LIN {X 0,Y 122.45,Z 109.011,A -85,B 0,C 180,E1 -25952.066,E2 -25952.066} C_VEL
LIN {X 0,Y 126.143,Z 114.519,A -85,B 0,C 180,E1 -25954.582,E2 -25954.582} C_VEL
LIN {X 0,Y 129.756,Z 120.065,A -85,B 0,C 180,E1 -25956.81,E2 -25956.81} C_VEL
LIN {X 0,Y 134.264,Z 129.772,A -85,B 0,C 180,E1 -25959.517,E2 -25959.517} C_VEL
LIN {X 0,Y 138.304,Z 140.286,A -85,B 0,C 180,E1 -25961.832,E2 -25961.832} C_VEL
LIN {X 0,Y 140.231,Z 146.487,A -85,B 0,C 180,E1 -25962.943,E2 -25962.943} C_VEL
LIN {X 0,Y 141.292,Z 167.319,A -85,B 0,C 180,E1 -25964.672,E2 -25964.672} C_VEL
LIN {X 0,Y 138.783,Z 203.821,A -85,B 0,C 180,E1 -25966.343,E2 -25966.343} C_VEL
LIN {X 0,Y 136.982,Z 217.471,A -85,B 0,C 180,E1 -25967.481,E2 -25967.481} C_VEL
LIN {X 0,Y 134.526,Z 229.675,A -85,B 0,C 180,E1 -25968.981,E2 -25968.981} C_VEL
LIN {X 0,Y 131.446,Z 241.678,A -85,B 0,C 180,E1 -25971.079,E2 -25971.079} C_VEL
LIN {X 0,Y 127.778,Z 253.16,A -85,B 0,C 180,E1 -25973.752,E2 -25973.752} C_VEL
LIN {X 0,Y 124.606,Z 262.476,A -85,B 0,C 180,E1 -25976.637,E2 -25976.637} C_VEL
LIN {X 0,Y 121.036,Z 272.287,A -85,B 0,C 180,E1 -25980.572,E2 -25980.572} C_VEL
LIN {X 0,Y 118.688,Z 278.374,A -85,B 0,C 180,E1 -25983.633,E2 -25983.633} C_VEL
LIN {X 0,Y 115.905,Z 286.343,A -85,B 0,C 180,E1 -25988.664,E2 -25988.664} C_VEL
LIN {X 0,Y 113.859,Z 292.673,A -85,B 0,C 180,E1 -25993.872,E2 -25993.872} C_VEL
LIN {X 0,Y 112.784,Z 297.7,A -85,B 0,C 180,E1 -25999.224,E2 -25999.224} C_VEL
LIN {X 0,Y 112.572,Z 301.563,A -85,B 0,C 180,E1 -26004.625,E2 -26004.625} C_VEL
LIN {X 0,Y 112.803,Z 304.341,A -85,B 0,C 180,E1 -26009.999,E2 -26009.999} C_VEL
LIN {X 0,Y 112.582,Z 305.583,A -85,B 0,C 180,E1 -26013.578,E2 -26013.578} C_VEL
LIN {X 0,Y 112.809,Z 306.873,A -85,B 0,C 180,E1 -26020.771,E2 -26020.771} C_VEL
LIN {X 0,Y 114.614,Z 306.557,A -85,B 0,C 180,E1 -26027.853,E2 -26027.853} C_VEL
LIN {X 0,Y 118.283,Z 304.747,A -85,B 0,C 180,E1 -26034.576,E2 -26034.576} C_VEL
LIN {X 0,Y 120.676,Z 303.239,A -85,B 0,C 180,E1 -26037.768,E2 -26037.768} C_VEL
LIN {X 0,Y 125.854,Z 299.488,A -85,B 0,C 180,E1 -26043.109,E2 -26043.109} C_VEL
LIN {X 0,Y 131.819,Z 294.518,A -85,B 0,C 180,E1 -26047.814,E2 -26047.814} C_VEL
LIN {X 0,Y 137.879,Z 288.943,A -85,B 0,C 180,E1 -26051.5,E2 -26051.5} C_VEL
LIN {X 0,Y 144.484,Z 282.029,A -85,B 0,C 180,E1 -26054.853,E2 -26054.853} C_VEL
LIN {X 0,Y 150.329,Z 275.005,A -85,B 0,C 180,E1 -26057.418,E2 -26057.418} C_VEL
LIN {X 0,Y 153.184,Z 271.302,A -85,B 0,C 180,E1 -26058.5,E2 -26058.5} C_VEL
LIN {X 0,Y 155.841,Z 267.217,A -85,B 0,C 180,E1 -26059.737,E2 -26059.737} C_VEL
LIN {X 0,Y 158.817,Z 260.366,A -85,B 0,C 180,E1 -26062.115,E2 -26062.115} C_VEL
LIN {X 0,Y 161.563,Z 253.029,A -85,B 0,C 180,E1 -26064.286,E2 -26064.286} C_VEL
LIN {X 0,Y 163.755,Z 248.186,A -85,B 0,C 180,E1 -26065.183,E2 -26065.183} C_VEL
LIN {X 0,Y 168.724,Z 237.706,A -85,B 0,C 180,E1 -26066.414,E2 -26066.414} C_VEL
LIN {X 0,Y 173.412,Z 225.079,A -85,B 0,C 180,E1 -26067.508,E2 -26067.508} C_VEL
LIN {X 0,Y 176.771,Z 212.767,A -85,B 0,C 180,E1 -26068.283,E2 -26068.283} C_VEL
LIN {X 0,Y 179.12,Z 199.548,A -85,B 0,C 180,E1 -26068.839,E2 -26068.839} C_VEL
LIN {X 0,Y 179.992,Z 191.121,A -85,B 0,C 180,E1 -26069.109,E2 -26069.109} C_VEL
LIN {X 0,Y 176.857,Z 181.807,A -85,B 0,C 180,E1 -26072.407,E2 -26072.407} C_VEL
LIN {X 0,Y 174.407,Z 175.318,A -85,B 0,C 180,E1 -26075.367,E2 -26075.367} C_VEL
LIN {X 0,Y 172.703,Z 171.191,A -85,B 0,C 180,E1 -26077.731,E2 -26077.731} C_VEL
LIN {X 0,Y 171.544,Z 168.304,A -85,B 0,C 180,E1 -26079.638,E2 -26079.638} C_VEL
LIN {X 0,Y 170.023,Z 164.562,A -85,B 0,C 180,E1 -26082.687,E2 -26082.687} C_VEL
LIN {X 0,Y 168.16,Z 160.166,A -85,B 0,C 180,E1 -26088.55,E2 -26088.55} C_VEL
LIN {X 0,Y 167.654,Z 159.81,A -85,B 0,C 180,E1 -26095.191,E2 -26095.191} C_VEL
LIN {X 0,Y 168.258,Z 159.961,A -85,B 0,C 180,E1 -26098.515,E2 -26098.515} C_VEL
LIN {X 0,Y 169.813,Z 163.596,A -85,B 0,C 180,E1 -26103.49,E2 -26103.49} C_VEL
LIN {X 0,Y 170.565,Z 164.869,A -85,B 0,C 180,E1 -26105.061,E2 -26105.061} C_VEL
LIN {X 0,Y 172.912,Z 169.191,A -85,B 0,C 180,E1 -26108.993,E2 -26108.993} C_VEL
LIN {X 0,Y 174.96,Z 172.997,A -85,B 0,C 180,E1 -26111.66,E2 -26111.66} C_VEL
LIN {X 0,Y 177.973,Z 178.76,A -85,B 0,C 180,E1 -26114.947,E2 -26114.947} C_VEL
LIN {X 0,Y 180.591,Z 184.208,A -85,B 0,C 180,E1 -26117.431,E2 -26117.431} C_VEL
LIN {X 0,Y 178.865,Z 198.313,A -85,B 0,C 180,E1 -26117.998,E2 -26117.998} C_VEL
LIN {X 0,Y 176.444,Z 209.589,A -85,B 0,C 180,E1 -26118.65,E2 -26118.65} C_VEL
LIN {X 0,Y 172.507,Z 222.682,A -85,B 0,C 180,E1 -26119.771,E2 -26119.771} C_VEL
LIN {X 0,Y 167.722,Z 234.725,A -85,B 0,C 180,E1 -26121.202,E2 -26121.202} C_VEL
LIN {X 0,Y 161.91,Z 246.089,A -85,B 0,C 180,E1 -26122.996,E2 -26122.996} C_VEL
LIN {X 0,Y 155.356,Z 256.599,A -85,B 0,C 180,E1 -26125.211,E2 -26125.211} C_VEL
LIN {X 0,Y 149.014,Z 265.155,A -85,B 0,C 180,E1 -26127.643,E2 -26127.643} C_VEL
LIN {X 0,Y 141.367,Z 273.791,A -85,B 0,C 180,E1 -26130.956,E2 -26130.956} C_VEL
LIN {X 0,Y 135.511,Z 279.488,A -85,B 0,C 180,E1 -26133.923,E2 -26133.923} C_VEL
LIN {X 0,Y 129.063,Z 284.989,A -85,B 0,C 180,E1 -26137.856,E2 -26137.856} C_VEL
LIN {X 0,Y 123.213,Z 289.225,A -85,B 0,C 180,E1 -26142.142,E2 -26142.142} C_VEL
LIN {X 0,Y 119.679,Z 291.431,A -85,B 0,C 180,E1 -26145.198,E2 -26145.198} C_VEL
LIN {X 0,Y 116.501,Z 293.121,A -85,B 0,C 180,E1 -26148.428,E2 -26148.428} C_VEL
LIN {X 0,Y 111.529,Z 295.153,A -85,B 0,C 180,E1 -26155.006,E2 -26155.006} C_VEL
LIN {X 0,Y 109.306,Z 295.609,A -85,B 0,C 180,E1 -26159.046,E2 -26159.046} C_VEL
LIN {X 0,Y 107.714,Z 295.578,A -85,B 0,C 180,E1 -26162.825,E2 -26162.825} C_VEL
LIN {X 0,Y 106.239,Z 294.936,A -85,B 0,C 180,E1 -26167.844,E2 -26167.844} C_VEL
LIN {X 0,Y 105.204,Z 293.009,A -85,B 0,C 180,E1 -26174.503,E2 -26174.503} C_VEL
LIN {X 0,Y 105.355,Z 290.275,A -85,B 0,C 180,E1 -26180.401,E2 -26180.401} C_VEL
LIN {X 0,Y 106.271,Z 286.516,A -85,B 0,C 180,E1 -26186.209,E2 -26186.209} C_VEL
LIN {X 0,Y 107.818,Z 281.647,A -85,B 0,C 180,E1 -26191.869,E2 -26191.869} C_VEL
LIN {X 0,Y 110.085,Z 275.523,A -85,B 0,C 180,E1 -26197.337,E2 -26197.337} C_VEL
LIN {X 0,Y 113.199,Z 267.91,A -85,B 0,C 180,E1 -26202.552,E2 -26202.552} C_VEL
LIN {X 0,Y 116.412,Z 260.121,A -85,B 0,C 180,E1 -26206.666,E2 -26206.666} C_VEL
LIN {X 0,Y 120.098,Z 250.61,A -85,B 0,C 180,E1 -26210.557,E2 -26210.557} C_VEL
LIN {X 0,Y 123.738,Z 240.071,A -85,B 0,C 180,E1 -26213.872,E2 -26213.872} C_VEL
LIN {X 0,Y 127.123,Z 228.378,A -85,B 0,C 180,E1 -26216.693,E2 -26216.693} C_VEL
LIN {X 0,Y 130.218,Z 215.809,A -85,B 0,C 180,E1 -26218.841,E2 -26218.841} C_VEL
LIN {X 0,Y 132.564,Z 202.695,A -85,B 0,C 180,E1 -26220.45,E2 -26220.45} C_VEL
LIN {X 0,Y 134.047,Z 189.846,A -85,B 0,C 180,E1 -26221.461,E2 -26221.461} C_VEL
LIN {X 0,Y 137.031,Z 146.864,A -85,B 0,C 180,E1 -26223.415,E2 -26223.415} C_VEL
LIN {X 0,Y 131.983,Z 135.808,A -85,B 0,C 180,E1 -26226.218,E2 -26226.218} C_VEL
LIN {X 0,Y 126.284,Z 125.434,A -85,B 0,C 180,E1 -26229.657,E2 -26229.657} C_VEL
LIN {X 0,Y 120.985,Z 117.374,A -85,B 0,C 180,E1 -26233.233,E2 -26233.233} C_VEL
LIN {X 0,Y 118.365,Z 113.693,A -85,B 0,C 180,E1 -26235.205,E2 -26235.205} C_VEL
LIN {X 0,Y 115.945,Z 110.284,A -85,B 0,C 180,E1 -26237.198,E2 -26237.198} C_VEL
LIN {X 0,Y 114.847,Z 109.03,A -85,B 0,C 180,E1 -26238.132,E2 -26238.132} C_VEL
LIN {X 0,Y 112.7,Z 106.255,A -85,B 0,C 180,E1 -26240.122,E2 -26240.122} C_VEL
LIN {X 0,Y 111.818,Z 104.593,A -85,B 0,C 180,E1 -26241.058,E2 -26241.058} C_VEL
LIN {X 0,Y 109.131,Z 102.466,A -85,B 0,C 180,E1 -26243.769,E2 -26243.769} C_VEL
LIN {X 0,Y 107.991,Z 100.283,A -85,B 0,C 180,E1 -26245.22,E2 -26245.22} C_VEL
LIN {X 0,Y 107.742,Z 98.998,A -85,B 0,C 180,E1 -26245.795,E2 -26245.795} C_VEL
LIN {X 0,Y 107.8,Z 99.021,A -85,B 0,C 180,E1 -26248.562,E2 -26248.562} C_VEL
LIN {X 0,Y 107.862,Z 99.029,A -85,B 0,C 180,E1 -26255.814,E2 -26255.814} C_VEL
LIN {X 0,Y 107.907,Z 99.037,A -85,B 0,C 180,E1 -26260.994,E2 -26260.994} C_VEL
LIN {X 0,Y 108.257,Z 98.997,A -85,B 0,C 180,E1 -26268.768,E2 -26268.768} C_VEL
LIN {X 0,Y 108.45,Z 98.975,A -85,B 0,C 180,E1 -26276.284,E2 -26276.284} C_VEL
LIN {X 0,Y 108.922,Z 98.897,A -85,B 0,C 180,E1 -26279.999,E2 -26279.999} C_VEL
LIN {X 0,Y 108.306,Z 98.976,A -85,B 0,C 180,E1 -26287.456,E2 -26287.456} C_VEL
LIN {X 0,Y 108.178,Z 99.006,A -85,B 0,C 180,E1 -26292.959,E2 -26292.959} C_VEL
LIN {X 0,Y 107.895,Z 99.064,A -85,B 0,C 180,E1 -26299.748,E2 -26299.748} C_VEL
LIN {X 0,Y 108.638,Z 101.364,A -85,B 0,C 180,E1 -26300.842,E2 -26300.842} C_VEL
LIN {X 0,Y 110.574,Z 103.726,A -85,B 0,C 180,E1 -26302.993,E2 -26302.993} C_VEL
LIN {X 0,Y 112.138,Z 104.975,A -85,B 0,C 180,E1 -26304.502,E2 -26304.502} C_VEL
LIN {X 0,Y 114.06,Z 108.164,A -85,B 0,C 180,E1 -26306.409,E2 -26306.409} C_VEL
LIN {X 0,Y 115.947,Z 110.168,A -85,B 0,C 180,E1 -26308.018,E2 -26308.018} C_VEL
LIN {X 0,Y 118.401,Z 113.66,A -85,B 0,C 180,E1 -26310.04,E2 -26310.04} C_VEL
LIN {X 0,Y 122.41,Z 119.495,A -85,B 0,C 180,E1 -26313.007,E2 -26313.007} C_VEL
LIN {X 0,Y 126.307,Z 125.87,A -85,B 0,C 180,E1 -26315.626,E2 -26315.626} C_VEL
LIN {X 0,Y 131.184,Z 137.371,A -85,B 0,C 180,E1 -26318.796,E2 -26318.796} C_VEL
LIN {X 0,Y 134.821,Z 148.268,A -85,B 0,C 180,E1 -26321.079,E2 -26321.079} C_VEL
LIN {X 0,Y 135.709,Z 164.102,A -85,B 0,C 180,E1 -26322.531,E2 -26322.531} C_VEL
LIN {X 0,Y 135.65,Z 169.911,A -85,B 0,C 180,E1 -26322.912,E2 -26322.912} C_VEL
LIN {X 0,Y 133.158,Z 204.005,A -85,B 0,C 180,E1 -26324.525,E2 -26324.525} C_VEL
LIN {X 0,Y 131.269,Z 217.462,A -85,B 0,C 180,E1 -26325.684,E2 -26325.684} C_VEL
LIN {X 0,Y 128.699,Z 229.567,A -85,B 0,C 180,E1 -26327.219,E2 -26327.219} C_VEL
LIN {X 0,Y 125.48,Z 241.506,A -85,B 0,C 180,E1 -26329.374,E2 -26329.374} C_VEL
LIN {X 0,Y 121.634,Z 252.948,A -85,B 0,C 180,E1 -26332.126,E2 -26332.126} C_VEL
LIN {X 0,Y 118.293,Z 262.236,A -85,B 0,C 180,E1 -26335.12,E2 -26335.12} C_VEL
LIN {X 0,Y 114.982,Z 270.896,A -85,B 0,C 180,E1 -26338.699,E2 -26338.699} C_VEL
LIN {X 0,Y 112.256,Z 277.325,A -85,B 0,C 180,E1 -26341.993,E2 -26341.993} C_VEL
LIN {X 0,Y 109.258,Z 285.443,A -85,B 0,C 180,E1 -26347.296,E2 -26347.296} C_VEL
LIN {X 0,Y 106.998,Z 291.889,A -85,B 0,C 180,E1 -26352.807,E2 -26352.807} C_VEL
LIN {X 0,Y 105.786,Z 297.003,A -85,B 0,C 180,E1 -26358.502,E2 -26358.502} C_VEL
LIN {X 0,Y 105.479,Z 300.944,A -85,B 0,C 180,E1 -26364.263,E2 -26364.263} C_VEL
LIN {X 0,Y 105.727,Z 303.8,A -85,B 0,C 180,E1 -26369.999,E2 -26369.999} C_VEL
LIN {X 0,Y 105.495,Z 305.076,A -85,B 0,C 180,E1 -26373.818,E2 -26373.818} C_VEL
LIN {X 0,Y 105.814,Z 306.437,A -85,B 0,C 180,E1 -26381.492,E2 -26381.492} C_VEL
LIN {X 0,Y 106.625,Z 306.536,A -85,B 0,C 180,E1 -26385.286,E2 -26385.286} C_VEL
LIN {X 0,Y 109.606,Z 305.539,A -85,B 0,C 180,E1 -26392.625,E2 -26392.625} C_VEL
LIN {X 0,Y 114.425,Z 303.036,A -85,B 0,C 180,E1 -26399.429,E2 -26399.429} C_VEL
LIN {X 0,Y 119.496,Z 299.708,A -85,B 0,C 180,E1 -26404.575,E2 -26404.575} C_VEL
LIN {X 0,Y 126.28,Z 294.491,A -85,B 0,C 180,E1 -26409.792,E2 -26409.792} C_VEL
LIN {X 0,Y 133.728,Z 287.998,A -85,B 0,C 180,E1 -26414.133,E2 -26414.133} C_VEL
LIN {X 0,Y 140.758,Z 280.932,A -85,B 0,C 180,E1 -26417.429,E2 -26417.429} C_VEL
LIN {X 0,Y 146.812,Z 273.785,A -85,B 0,C 180,E1 -26419.988,E2 -26419.988} C_VEL
LIN {X 0,Y 150.768,Z 268.778,A -85,B 0,C 180,E1 -26421.332,E2 -26421.332} C_VEL
LIN {X 0,Y 157.429,Z 259.05,A -85,B 0,C 180,E1 -26423.47,E2 -26423.47} C_VEL
LIN {X 0,Y 163.755,Z 248.186,A -85,B 0,C 180,E1 -26425.183,E2 -26425.183} C_VEL
LIN {X 0,Y 165.904,Z 243.232,A -85,B 0,C 180,E1 -26426.011,E2 -26426.011} C_VEL
LIN {X 0,Y 168.222,Z 234.981,A -85,B 0,C 180,E1 -26427.743,E2 -26427.743} C_VEL
LIN {X 0,Y 170.157,Z 226.466,A -85,B 0,C 180,E1 -26429.33,E2 -26429.33} C_VEL
LIN {X 0,Y 171.563,Z 221.002,A -85,B 0,C 180,E1 -26429.914,E2 -26429.914} C_VEL
LIN {X 0,Y 174.755,Z 208.28,A -85,B 0,C 180,E1 -26430.575,E2 -26430.575} C_VEL
LIN {X 0,Y 176.771,Z 195.011,A -85,B 0,C 180,E1 -26431.061,E2 -26431.061} C_VEL
LIN {X 0,Y 176.717,Z 193.931,A -85,B 0,C 180,E1 -26431.218,E2 -26431.218} C_VEL
LIN {X 0,Y 174.265,Z 186.165,A -85,B 0,C 180,E1 -26434.148,E2 -26434.148} C_VEL
LIN {X 0,Y 171.921,Z 179.559,A -85,B 0,C 180,E1 -26437.386,E2 -26437.386} C_VEL
LIN {X 0,Y 170.006,Z 174.486,A -85,B 0,C 180,E1 -26440.688,E2 -26440.688} C_VEL
LIN {X 0,Y 168.773,Z 171.173,A -85,B 0,C 180,E1 -26443.438,E2 -26443.438} C_VEL
LIN {X 0,Y 167.156,Z 167.137,A -85,B 0,C 180,E1 -26449.094,E2 -26449.094} C_VEL
LIN {X 0,Y 166.773,Z 166.854,A -85,B 0,C 180,E1 -26455.166,E2 -26455.166} C_VEL
LIN {X 0,Y 167.29,Z 167.015,A -85,B 0,C 180,E1 -26458.195,E2 -26458.195} C_VEL
LIN {X 0,Y 168.981,Z 170.859,A -85,B 0,C 180,E1 -26463.652,E2 -26463.652} C_VEL
LIN {X 0,Y 171.441,Z 175.774,A -85,B 0,C 180,E1 -26468.246,E2 -26468.246} C_VEL
LIN {X 0,Y 173.46,Z 179.789,A -85,B 0,C 180,E1 -26471.065,E2 -26471.065} C_VEL
LIN {X 0,Y 176.181,Z 185.405,A -85,B 0,C 180,E1 -26474.217,E2 -26474.217} C_VEL
LIN {X 0,Y 177.361,Z 187.99,A -85,B 0,C 180,E1 -26475.453,E2 -26475.453} C_VEL
LIN {X 0,Y 175.483,Z 200.905,A -85,B 0,C 180,E1 -26476.019,E2 -26476.019} C_VEL
LIN {X 0,Y 172.389,Z 213.819,A -85,B 0,C 180,E1 -26476.836,E2 -26476.836} C_VEL
LIN {X 0,Y 168.838,Z 224.584,A -85,B 0,C 180,E1 -26477.793,E2 -26477.793} C_VEL
LIN {X 0,Y 164.475,Z 235.023,A -85,B 0,C 180,E1 -26479.024,E2 -26479.024} C_VEL
LIN {X 0,Y 158.413,Z 246.497,A -85,B 0,C 180,E1 -26480.789,E2 -26480.789} C_VEL
LIN {X 0,Y 152.365,Z 255.923,A -85,B 0,C 180,E1 -26482.705,E2 -26482.705} C_VEL
LIN {X 0,Y 145.42,Z 265.067,A -85,B 0,C 180,E1 -26485.185,E2 -26485.185} C_VEL
LIN {X 0,Y 137.722,Z 273.511,A -85,B 0,C 180,E1 -26488.327,E2 -26488.327} C_VEL
LIN {X 0,Y 130.352,Z 280.348,A -85,B 0,C 180,E1 -26491.864,E2 -26491.864} C_VEL
LIN {X 0,Y 122.493,Z 286.54,A -85,B 0,C 180,E1 -26496.561,E2 -26496.561} C_VEL
LIN {X 0,Y 116.238,Z 290.588,A -85,B 0,C 180,E1 -26501.173,E2 -26501.173} C_VEL
LIN {X 0,Y 111.063,Z 293.32,A -85,B 0,C 180,E1 -26505.889,E2 -26505.889} C_VEL
LIN {X 0,Y 107.996,Z 294.627,A -85,B 0,C 180,E1 -26509.403,E2 -26509.403} C_VEL
LIN {X 0,Y 105.137,Z 295.571,A -85,B 0,C 180,E1 -26513.338,E2 -26513.338} C_VEL
LIN {X 0,Y 103.036,Z 295.986,A -85,B 0,C 180,E1 -26516.931,E2 -26516.931} C_VEL
LIN {X 0,Y 101.203,Z 295.999,A -85,B 0,C 180,E1 -26520.916,E2 -26520.916} C_VEL
LIN {X 0,Y 99.311,Z 295.302,A -85,B 0,C 180,E1 -26526.926,E2 -26526.926} C_VEL
LIN {X 0,Y 98.2,Z 293.605,A -85,B 0,C 180,E1 -26533.367,E2 -26533.367} C_VEL
LIN {X 0,Y 98.203,Z 290.964,A -85,B 0,C 180,E1 -26539.695,E2 -26539.695} C_VEL
LIN {X 0,Y 99.067,Z 287.302,A -85,B 0,C 180,E1 -26545.933,E2 -26545.933} C_VEL
LIN {X 0,Y 100.652,Z 282.536,A -85,B 0,C 180,E1 -26552.002,E2 -26552.002} C_VEL
LIN {X 0,Y 103.508,Z 275.394,A -85,B 0,C 180,E1 -26558.789,E2 -26558.789} C_VEL
LIN {X 0,Y 106.897,Z 267.646,A -85,B 0,C 180,E1 -26564.275,E2 -26564.275} C_VEL
LIN {X 0,Y 111.091,Z 257.912,A -85,B 0,C 180,E1 -26569.4,E2 -26569.4} C_VEL
LIN {X 0,Y 114.979,Z 248.275,A -85,B 0,C 180,E1 -26573.231,E2 -26573.231} C_VEL
LIN {X 0,Y 118.574,Z 237.94,A -85,B 0,C 180,E1 -26576.395,E2 -26576.395} C_VEL
LIN {X 0,Y 121.788,Z 227.166,A -85,B 0,C 180,E1 -26578.902,E2 -26578.902} C_VEL
LIN {X 0,Y 125.023,Z 214.295,A -85,B 0,C 180,E1 -26581.064,E2 -26581.064} C_VEL
LIN {X 0,Y 127.273,Z 201.737,A -85,B 0,C 180,E1 -26582.559,E2 -26582.559} C_VEL
LIN {X 0,Y 128.774,Z 188.552,A -85,B 0,C 180,E1 -26583.549,E2 -26583.549} C_VEL
LIN {X 0,Y 131.641,Z 149.15,A -85,B 0,C 180,E1 -26585.36,E2 -26585.36} C_VEL
LIN {X 0,Y 127.505,Z 139.82,A -85,B 0,C 180,E1 -26587.888,E2 -26587.888} C_VEL
LIN {X 0,Y 122.374,Z 130.243,A -85,B 0,C 180,E1 -26591.267,E2 -26591.267} C_VEL
LIN {X 0,Y 117.394,Z 122.443,A -85,B 0,C 180,E1 -26594.95,E2 -26594.95} C_VEL
LIN {X 0,Y 115.094,Z 119.173,A -85,B 0,C 180,E1 -26596.842,E2 -26596.842} C_VEL
LIN {X 0,Y 112.326,Z 115.229,A -85,B 0,C 180,E1 -26599.356,E2 -26599.356} C_VEL
LIN {X 0,Y 109.902,Z 111.933,A -85,B 0,C 180,E1 -26601.797,E2 -26601.797} C_VEL
LIN {X 0,Y 109.106,Z 110.795,A -85,B 0,C 180,E1 -26602.668,E2 -26602.668} C_VEL
LIN {X 0,Y 106.527,Z 108.161,A -85,B 0,C 180,E1 -26605.603,E2 -26605.603} C_VEL
LIN {X 0,Y 105.263,Z 105.654,A -85,B 0,C 180,E1 -26607.405,E2 -26607.405} C_VEL
LIN {X 0,Y 102.502,Z 103.847,A -85,B 0,C 180,E1 -26611.316,E2 -26611.316} C_VEL
LIN {X 0,Y 101.086,Z 101.44,A -85,B 0,C 180,E1 -26614.051,E2 -26614.051} C_VEL
LIN {X 0,Y 100.778,Z 99.911,A -85,B 0,C 180,E1 -26615.041,E2 -26615.041} C_VEL
LIN {X 0,Y 100.819,Z 99.927,A -85,B 0,C 180,E1 -26619.601,E2 -26619.601} C_VEL
LIN {X 0,Y 101.105,Z 99.885,A -85,B 0,C 180,E1 -26626.702,E2 -26626.702} C_VEL
LIN {X 0,Y 101.246,Z 99.851,A -85,B 0,C 180,E1 -26632.019,E2 -26632.019} C_VEL
LIN {X 0,Y 101.849,Z 99.777,A -85,B 0,C 180,E1 -26639.999,E2 -26639.999} C_VEL
LIN {X 0,Y 101.185,Z 99.869,A -85,B 0,C 180,E1 -26649.999,E2 -26649.999} C_VEL
LIN {X 0,Y 101.236,Z 100.081,A -85,B 0,C 180,E1 -26651.132,E2 -26651.132} C_VEL
LIN {X 0,Y 102.055,Z 102.596,A -85,B 0,C 180,E1 -26652.993,E2 -26652.993} C_VEL
LIN {X 0,Y 103.861,Z 104.818,A -85,B 0,C 180,E1 -26655.955,E2 -26655.955} C_VEL
LIN {X 0,Y 105.624,Z 105.943,A -85,B 0,C 180,E1 -26658.298,E2 -26658.298} C_VEL
LIN {X 0,Y 107.419,Z 109.132,A -85,B 0,C 180,E1 -26660.714,E2 -26660.714} C_VEL
LIN {X 0,Y 109.644,Z 111.32,A -85,B 0,C 180,E1 -26663.138,E2 -26663.138} C_VEL
LIN {X 0,Y 112.069,Z 114.908,A -85,B 0,C 180,E1 -26665.636,E2 -26665.636} C_VEL
LIN {X 0,Y 113.338,Z 116.523,A -85,B 0,C 180,E1 -26666.808,E2 -26666.808} C_VEL
LIN {X 0,Y 116.649,Z 121.303,A -85,B 0,C 180,E1 -26669.673,E2 -26669.673} C_VEL
LIN {X 0,Y 120.826,Z 127.796,A -85,B 0,C 180,E1 -26672.874,E2 -26672.874} C_VEL
LIN {X 0,Y 123.279,Z 132.744,A -85,B 0,C 180,E1 -26674.663,E2 -26674.663} C_VEL
LIN {X 0,Y 127.416,Z 143.33,A -85,B 0,C 180,E1 -26677.587,E2 -26677.587} C_VEL
LIN {X 0,Y 129.836,Z 151.229,A -85,B 0,C 180,E1 -26679.276,E2 -26679.276} C_VEL
LIN {X 0,Y 130.459,Z 168.381,A -85,B 0,C 180,E1 -26680.823,E2 -26680.823} C_VEL
LIN {X 0,Y 127.814,Z 203.093,A -85,B 0,C 180,E1 -26682.475,E2 -26682.475} C_VEL
LIN {X 0,Y 125.751,Z 217.127,A -85,B 0,C 180,E1 -26683.691,E2 -26683.691} C_VEL
LIN {X 0,Y 123.006,Z 229.451,A -85,B 0,C 180,E1 -26685.292,E2 -26685.292} C_VEL
LIN {X 0,Y 119.638,Z 241.334,A -85,B 0,C 180,E1 -26687.501,E2 -26687.501} C_VEL
LIN {X 0,Y 115.598,Z 252.736,A -85,B 0,C 180,E1 -26690.328,E2 -26690.328} C_VEL
LIN {X 0,Y 112.071,Z 261.996,A -85,B 0,C 180,E1 -26693.433,E2 -26693.433} C_VEL
LIN {X 0,Y 108.774,Z 270.085,A -85,B 0,C 180,E1 -26696.908,E2 -26696.908} C_VEL
LIN {X 0,Y 105.856,Z 276.54,A -85,B 0,C 180,E1 -26700.321,E2 -26700.321} C_VEL
LIN {X 0,Y 102.691,Z 284.516,A -85,B 0,C 180,E1 -26705.754,E2 -26705.754} C_VEL
LIN {X 0,Y 100.195,Z 291.093,A -85,B 0,C 180,E1 -26711.599,E2 -26711.599} C_VEL
LIN {X 0,Y 98.781,Z 296.302,A -85,B 0,C 180,E1 -26717.674,E2 -26717.674} C_VEL
LIN {X 0,Y 98.4,Z 300.326,A -85,B 0,C 180,E1 -26723.848,E2 -26723.848} C_VEL
LIN {X 0,Y 98.648,Z 303.253,A -85,B 0,C 180,E1 -26729.999,E2 -26729.999} C_VEL
LIN {X 0,Y 98.422,Z 304.57,A -85,B 0,C 180,E1 -26734.093,E2 -26734.093} C_VEL
LIN {X 0,Y 98.848,Z 305.998,A -85,B 0,C 180,E1 -26742.314,E2 -26742.314} C_VEL
LIN {X 0,Y 99.748,Z 306.146,A -85,B 0,C 180,E1 -26746.368,E2 -26746.368} C_VEL
LIN {X 0,Y 101.116,Z 305.887,A -85,B 0,C 180,E1 -26750.334,E2 -26750.334} C_VEL
LIN {X 0,Y 105.472,Z 304.22,A -85,B 0,C 180,E1 -26757.802,E2 -26757.802} C_VEL
LIN {X 0,Y 108.282,Z 302.817,A -85,B 0,C 180,E1 -26761.279,E2 -26761.279} C_VEL
LIN {X 0,Y 113.263,Z 299.851,A -85,B 0,C 180,E1 -26766.231,E2 -26766.231} C_VEL
LIN {X 0,Y 118.83,Z 296.007,A -85,B 0,C 180,E1 -26770.583,E2 -26770.583} C_VEL
LIN {X 0,Y 125.28,Z 291.018,A -85,B 0,C 180,E1 -26774.524,E2 -26774.524} C_VEL
LIN {X 0,Y 132.342,Z 284.786,A -85,B 0,C 180,E1 -26778.026,E2 -26778.026} C_VEL
LIN {X 0,Y 139.841,Z 277.064,A -85,B 0,C 180,E1 -26781.166,E2 -26781.166} C_VEL
LIN {X 0,Y 143.762,Z 272.504,A -85,B 0,C 180,E1 -26782.597,E2 -26782.597} C_VEL
LIN {X 0,Y 149.149,Z 265.629,A -85,B 0,C 180,E1 -26784.372,E2 -26784.372} C_VEL
LIN {X 0,Y 156.17,Z 255.198,A -85,B 0,C 180,E1 -26786.359,E2 -26786.359} C_VEL
LIN {X 0,Y 162.7,Z 243.478,A -85,B 0,C 180,E1 -26787.963,E2 -26787.963} C_VEL
LIN {X 0,Y 167.895,Z 231.763,A -85,B 0,C 180,E1 -26789.104,E2 -26789.104} C_VEL
LIN {X 0,Y 171.563,Z 221.002,A -85,B 0,C 180,E1 -26789.914,E2 -26789.914} C_VEL
LIN {X 0,Y 172.342,Z 217.297,A -85,B 0,C 180,E1 -26790.351,E2 -26790.351} C_VEL
LIN {X 0,Y 172.774,Z 205.72,A -85,B 0,C 180,E1 -26792.663,E2 -26792.663} C_VEL
LIN {X 0,Y 173.183,Z 201.902,A -85,B 0,C 180,E1 -26793.001,E2 -26793.001} C_VEL
LIN {X 0,Y 173.791,Z 197.441,A -85,B 0,C 180,E1 -26793.171,E2 -26793.171} C_VEL
LIN {X 0,Y 171.677,Z 190.161,A -85,B 0,C 180,E1 -26796.156,E2 -26796.156} C_VEL
LIN {X 0,Y 169.892,Z 184.799,A -85,B 0,C 180,E1 -26799.018,E2 -26799.018} C_VEL
LIN {X 0,Y 168.649,Z 181.093,A -85,B 0,C 180,E1 -26801.473,E2 -26801.473} C_VEL
LIN {X 0,Y 167.529,Z 177.762,A -85,B 0,C 180,E1 -26804.257,E2 -26804.257} C_VEL
LIN {X 0,Y 166.195,Z 174.134,A -85,B 0,C 180,E1 -26809.493,E2 -26809.493} C_VEL
LIN {X 0,Y 165.892,Z 173.898,A -85,B 0,C 180,E1 -26815.14,E2 -26815.14} C_VEL
LIN {X 0,Y 166.331,Z 174.071,A -85,B 0,C 180,E1 -26817.882,E2 -26817.882} C_VEL
LIN {X 0,Y 168.033,Z 178.165,A -85,B 0,C 180,E1 -26823.613,E2 -26823.613} C_VEL
LIN {X 0,Y 170.07,Z 182.477,A -85,B 0,C 180,E1 -26827.597,E2 -26827.597} C_VEL
LIN {X 0,Y 172.417,Z 187.468,A -85,B 0,C 180,E1 -26831.029,E2 -26831.029} C_VEL
LIN {X 0,Y 174.312,Z 191.904,A -85,B 0,C 180,E1 -26833.45,E2 -26833.45} C_VEL
LIN {X 0,Y 172.032,Z 204.811,A -85,B 0,C 180,E1 -26834.039,E2 -26834.039} C_VEL
LIN {X 0,Y 168.632,Z 217.274,A -85,B 0,C 180,E1 -26834.901,E2 -26834.901} C_VEL
LIN {X 0,Y 164.463,Z 228.573,A -85,B 0,C 180,E1 -26835.955,E2 -26835.955} C_VEL
LIN {X 0,Y 159.225,Z 239.751,A -85,B 0,C 180,E1 -26837.354,E2 -26837.354} C_VEL
LIN {X 0,Y 153.272,Z 249.955,A -85,B 0,C 180,E1 -26839.028,E2 -26839.028} C_VEL
LIN {X 0,Y 146.804,Z 259.144,A -85,B 0,C 180,E1 -26841.011,E2 -26841.011} C_VEL
LIN {X 0,Y 139.803,Z 267.568,A -85,B 0,C 180,E1 -26843.448,E2 -26843.448} C_VEL
LIN {X 0,Y 131.737,Z 275.752,A -85,B 0,C 180,E1 -26846.675,E2 -26846.675} C_VEL
LIN {X 0,Y 125.349,Z 281.231,A -85,B 0,C 180,E1 -26849.655,E2 -26849.655} C_VEL
LIN {X 0,Y 118.226,Z 286.534,A -85,B 0,C 180,E1 -26853.673,E2 -26853.673} C_VEL
LIN {X 0,Y 111.703,Z 290.583,A -85,B 0,C 180,E1 -26858.147,E2 -26858.147} C_VEL
LIN {X 0,Y 105.882,Z 293.516,A -85,B 0,C 180,E1 -26863.105,E2 -26863.105} C_VEL
LIN {X 0,Y 102.487,Z 294.872,A -85,B 0,C 180,E1 -26866.708,E2 -26866.708} C_VEL
LIN {X 0,Y 98.803,Z 295.997,A -85,B 0,C 180,E1 -26871.487,E2 -26871.487} C_VEL
LIN {X 0,Y 94.822,Z 296.42,A -85,B 0,C 180,E1 -26878.748,E2 -26878.748} C_VEL
LIN {X 0,Y 92.386,Z 295.659,A -85,B 0,C 180,E1 -26885.908,E2 -26885.908} C_VEL
LIN {X 0,Y 91.222,Z 294.195,A -85,B 0,C 180,E1 -26892.053,E2 -26892.053} C_VEL
LIN {X 0,Y 91.05,Z 291.639,A -85,B 0,C 180,E1 -26898.875,E2 -26898.875} C_VEL
LIN {X 0,Y 91.872,Z 288.066,A -85,B 0,C 180,E1 -26905.614,E2 -26905.614} C_VEL
LIN {X 0,Y 93.488,Z 283.405,A -85,B 0,C 180,E1 -26912.156,E2 -26912.156} C_VEL
LIN {X 0,Y 96.437,Z 276.377,A -85,B 0,C 180,E1 -26919.439,E2 -26919.439} C_VEL
LIN {X 0,Y 99.981,Z 268.781,A -85,B 0,C 180,E1 -26925.285,E2 -26925.285} C_VEL
LIN {X 0,Y 103.628,Z 261.013,A -85,B 0,C 180,E1 -26929.823,E2 -26929.823} C_VEL
LIN {X 0,Y 108.024,Z 250.863,A -85,B 0,C 180,E1 -26934.317,E2 -26934.317} C_VEL
LIN {X 0,Y 111.839,Z 241.031,A -85,B 0,C 180,E1 -26937.611,E2 -26937.611} C_VEL
LIN {X 0,Y 115.623,Z 229.391,A -85,B 0,C 180,E1 -26940.603,E2 -26940.603} C_VEL
LIN {X 0,Y 119.066,Z 216.901,A -85,B 0,C 180,E1 -26942.842,E2 -26942.842} C_VEL
LIN {X 0,Y 121.681,Z 203.81,A -85,B 0,C 180,E1 -26944.525,E2 -26944.525} C_VEL
LIN {X 0,Y 123.392,Z 190.595,A -85,B 0,C 180,E1 -26945.611,E2 -26945.611} C_VEL
LIN {X 0,Y 126.45,Z 151.419,A -85,B 0,C 180,E1 -26947.44,E2 -26947.44} C_VEL
LIN {X 0,Y 122.573,Z 142.83,A -85,B 0,C 180,E1 -26950.049,E2 -26950.049} C_VEL
LIN {X 0,Y 118.343,Z 134.709,A -85,B 0,C 180,E1 -26953.151,E2 -26953.151} C_VEL
LIN {X 0,Y 113.774,Z 127.291,A -85,B 0,C 180,E1 -26956.899,E2 -26956.899} C_VEL
LIN {X 0,Y 109.706,Z 121.267,A -85,B 0,C 180,E1 -26960.787,E2 -26960.787} C_VEL
LIN {X 0,Y 107.199,Z 117.581,A -85,B 0,C 180,E1 -26963.563,E2 -26963.563} C_VEL
LIN {X 0,Y 104.093,Z 113.93,A -85,B 0,C 180,E1 -26967.445,E2 -26967.445} C_VEL
LIN {X 0,Y 103.117,Z 112.171,A -85,B 0,C 180,E1 -26968.946,E2 -26968.946} C_VEL
LIN {X 0,Y 100.582,Z 110.116,A -85,B 0,C 180,E1 -26972.987,E2 -26972.987} C_VEL
LIN {X 0,Y 99.13,Z 107,A -85,B 0,C 180,E1 -26976.317,E2 -26976.317} C_VEL
LIN {X 0,Y 95.676,Z 104.412,A -85,B 0,C 180,E1 -26989.417,E2 -26989.417} C_VEL
LIN {X 0,Y 95.703,Z 104.164,A -85,B 0,C 180,E1 -26995.788,E2 -26995.788} C_VEL
LIN {X 0,Y 96.419,Z 104.489,A -85,B 0,C 180,E1 -27000.521,E2 -27000.521} C_VEL
LIN {X 0,Y 98.398,Z 106.364,A -85,B 0,C 180,E1 -27007.179,E2 -27007.179} C_VEL
LIN {X 0,Y 99.524,Z 106.905,A -85,B 0,C 180,E1 -27009.654,E2 -27009.654} C_VEL
LIN {X 0,Y 100.878,Z 109.993,A -85,B 0,C 180,E1 -27012.69,E2 -27012.69} C_VEL
LIN {X 0,Y 103.151,Z 112.157,A -85,B 0,C 180,E1 -27016.322,E2 -27016.322} C_VEL
LIN {X 0,Y 103.849,Z 113.043,A -85,B 0,C 180,E1 -27017.348,E2 -27017.348} C_VEL
LIN {X 0,Y 106.153,Z 116.429,A -85,B 0,C 180,E1 -27020.465,E2 -27020.465} C_VEL
LIN {X 0,Y 107.306,Z 117.717,A -85,B 0,C 180,E1 -27021.806,E2 -27021.806} C_VEL
LIN {X 0,Y 110.793,Z 122.8,A -85,B 0,C 180,E1 -27025.547,E2 -27025.547} C_VEL
LIN {X 0,Y 114.567,Z 128.446,A -85,B 0,C 180,E1 -27029.012,E2 -27029.012} C_VEL
LIN {X 0,Y 118.364,Z 135.002,A -85,B 0,C 180,E1 -27032.116,E2 -27032.116} C_VEL
LIN {X 0,Y 122.512,Z 145.75,A -85,B 0,C 180,E1 -27035.398,E2 -27035.398} C_VEL
LIN {X 0,Y 124.836,Z 153.591,A -85,B 0,C 180,E1 -27037.211,E2 -27037.211} C_VEL
LIN {X 0,Y 125.224,Z 169.624,A -85,B 0,C 180,E1 -27038.69,E2 -27038.69} C_VEL
LIN {X 0,Y 122.479,Z 203.424,A -85,B 0,C 180,E1 -27040.345,E2 -27040.345} C_VEL
LIN {X 0,Y 120.349,Z 217.072,A -85,B 0,C 180,E1 -27041.563,E2 -27041.563} C_VEL
LIN {X 0,Y 117.465,Z 229.281,A -85,B 0,C 180,E1 -27043.18,E2 -27043.18} C_VEL
LIN {X 0,Y 113.937,Z 241.126,A -85,B 0,C 180,E1 -27045.439,E2 -27045.439} C_VEL
LIN {X 0,Y 109.689,Z 252.496,A -85,B 0,C 180,E1 -27048.335,E2 -27048.335} C_VEL
LIN {X 0,Y 105.956,Z 261.734,A -85,B 0,C 180,E1 -27051.548,E2 -27051.548} C_VEL
LIN {X 0,Y 102.123,Z 270.523,A -85,B 0,C 180,E1 -27055.525,E2 -27055.525} C_VEL
LIN {X 0,Y 99.011,Z 277.048,A -85,B 0,C 180,E1 -27059.263,E2 -27059.263} C_VEL
LIN {X 0,Y 95.683,Z 284.829,A -85,B 0,C 180,E1 -27065.016,E2 -27065.016} C_VEL
LIN {X 0,Y 93.445,Z 290.264,A -85,B 0,C 180,E1 -27070.216,E2 -27070.216} C_VEL
LIN {X 0,Y 91.812,Z 295.576,A -85,B 0,C 180,E1 -27076.722,E2 -27076.722} C_VEL
LIN {X 0,Y 91.318,Z 299.685,A -85,B 0,C 180,E1 -27083.369,E2 -27083.369} C_VEL
LIN {X 0,Y 91.553,Z 302.679,A -85,B 0,C 180,E1 -27089.998,E2 -27089.998} C_VEL
LIN {X 0,Y 91.352,Z 304.061,A -85,B 0,C 180,E1 -27094.411,E2 -27094.411} C_VEL
LIN {X 0,Y 91.914,Z 305.558,A -85,B 0,C 180,E1 -27103.259,E2 -27103.259} C_VEL
LIN {X 0,Y 94.459,Z 305.547,A -85,B 0,C 180,E1 -27111.838,E2 -27111.838} C_VEL
LIN {X 0,Y 99.213,Z 303.961,A -85,B 0,C 180,E1 -27119.725,E2 -27119.725} C_VEL
LIN {X 0,Y 105.669,Z 300.835,A -85,B 0,C 180,E1 -27126.767,E2 -27126.767} C_VEL
LIN {X 0,Y 111.424,Z 297.348,A -85,B 0,C 180,E1 -27131.472,E2 -27131.472} C_VEL
LIN {X 0,Y 117.989,Z 292.821,A -85,B 0,C 180,E1 -27135.623,E2 -27135.623} C_VEL
LIN {X 0,Y 126.451,Z 286.026,A -85,B 0,C 180,E1 -27139.834,E2 -27139.834} C_VEL
LIN {X 0,Y 134.197,Z 278.676,A -85,B 0,C 180,E1 -27143,E2 -27143} C_VEL
LIN {X 0,Y 139.57,Z 272.855,A -85,B 0,C 180,E1 -27144.909,E2 -27144.909} C_VEL
LIN {X 0,Y 146.613,Z 264.178,A -85,B 0,C 180,E1 -27147.019,E2 -27147.019} C_VEL
LIN {X 0,Y 153.861,Z 253.527,A -85,B 0,C 180,E1 -27148.919,E2 -27148.919} C_VEL
LIN {X 0,Y 159.827,Z 242.956,A -85,B 0,C 180,E1 -27150.278,E2 -27150.278} C_VEL
LIN {X 0,Y 165.15,Z 231.191,A -85,B 0,C 180,E1 -27151.364,E2 -27151.364} C_VEL
LIN {X 0,Y 169.626,Z 217.857,A -85,B 0,C 180,E1 -27152.305,E2 -27152.305} C_VEL
LIN {X 0,Y 172.681,Z 204.946,A -85,B 0,C 180,E1 -27152.888,E2 -27152.888} C_VEL
LIN {X 0,Y 173.183,Z 201.902,A -85,B 0,C 180,E1 -27153.001,E2 -27153.001} C_VEL
LIN {X 0,Y 173.266,Z 199.766,A -85,B 0,C 180,E1 -27153.308,E2 -27153.308} C_VEL
LIN {X 0,Y 172.794,Z 197.796,A -85,B 0,C 180,E1 -27154.074,E2 -27154.074} C_VEL
LIN {X 0,Y 171.634,Z 196.146,A -85,B 0,C 180,E1 -27155.453,E2 -27155.453} C_VEL
LIN {X 0,Y 169.593,Z 194.4,A -85,B 0,C 180,E1 -27157.876,E2 -27157.876} C_VEL
LIN {X 0,Y 168.768,Z 192.368,A -85,B 0,C 180,E1 -27159.214,E2 -27159.214} C_VEL
LIN {X 0,Y 167.264,Z 187.482,A -85,B 0,C 180,E1 -27162.423,E2 -27162.423} C_VEL
LIN {X 0,Y 166.305,Z 184.325,A -85,B 0,C 180,E1 -27165.127,E2 -27165.127} C_VEL
LIN {X 0,Y 165.316,Z 181.256,A -85,B 0,C 180,E1 -27169.436,E2 -27169.436} C_VEL
LIN {X 0,Y 165.011,Z 180.942,A -85,B 0,C 180,E1 -27175.114,E2 -27175.114} C_VEL
LIN {X 0,Y 165.394,Z 181.252,A -85,B 0,C 180,E1 -27177.717,E2 -27177.717} C_VEL
LIN {X 0,Y 166.919,Z 185.123,A -85,B 0,C 180,E1 -27183.168,E2 -27183.168} C_VEL
LIN {X 0,Y 168.757,Z 189.331,A -85,B 0,C 180,E1 -27187.027,E2 -27187.027} C_VEL
LIN {X 0,Y 170.697,Z 194.059,A -85,B 0,C 180,E1 -27190.299,E2 -27190.299} C_VEL
LIN {X 0,Y 171.35,Z 195.847,A -85,B 0,C 180,E1 -27191.362,E2 -27191.362} C_VEL
LIN {X 0,Y 168.684,Z 208.738,A -85,B 0,C 180,E1 -27192.024,E2 -27192.024} C_VEL
LIN {X 0,Y 164.931,Z 220.997,A -85,B 0,C 180,E1 -27192.909,E2 -27192.909} C_VEL
LIN {X 0,Y 160.27,Z 232.343,A -85,B 0,C 180,E1 -27194.027,E2 -27194.027} C_VEL
LIN {X 0,Y 154.122,Z 244.102,A -85,B 0,C 180,E1 -27195.573,E2 -27195.573} C_VEL
LIN {X 0,Y 147.308,Z 254.571,A -85,B 0,C 180,E1 -27197.413,E2 -27197.413} C_VEL
LIN {X 0,Y 139.924,Z 263.904,A -85,B 0,C 180,E1 -27199.654,E2 -27199.654} C_VEL
LIN {X 0,Y 132.306,Z 271.988,A -85,B 0,C 180,E1 -27202.287,E2 -27202.287} C_VEL
LIN {X 0,Y 124.495,Z 278.978,A -85,B 0,C 180,E1 -27205.417,E2 -27205.417} C_VEL
LIN {X 0,Y 116.308,Z 285.144,A -85,B 0,C 180,E1 -27209.451,E2 -27209.451} C_VEL
LIN {X 0,Y 109.554,Z 289.396,A -85,B 0,C 180,E1 -27213.495,E2 -27213.495} C_VEL
LIN {X 0,Y 104.06,Z 292.284,A -85,B 0,C 180,E1 -27217.435,E2 -27217.435} C_VEL
LIN {X 0,Y 97.223,Z 295.117,A -85,B 0,C 180,E1 -27223.71,E2 -27223.71} C_VEL
LIN {X 0,Y 92.611,Z 296.414,A -85,B 0,C 180,E1 -27229.367,E2 -27229.367} C_VEL
LIN {X 0,Y 88.584,Z 296.837,A -85,B 0,C 180,E1 -27236.267,E2 -27236.267} C_VEL
LIN {X 0,Y 85.511,Z 296.02,A -85,B 0,C 180,E1 -27244.701,E2 -27244.701} C_VEL
LIN {X 0,Y 84.316,Z 294.753,A -85,B 0,C 180,E1 -27250.526,E2 -27250.526} C_VEL
LIN {X 0,Y 83.903,Z 293.216,A -85,B 0,C 180,E1 -27255.448,E2 -27255.448} C_VEL
LIN {X 0,Y 84.292,Z 290.079,A -85,B 0,C 180,E1 -27262.82,E2 -27262.82} C_VEL
LIN {X 0,Y 85.661,Z 285.885,A -85,B 0,C 180,E1 -27270.002,E2 -27270.002} C_VEL
LIN {X 0,Y 88.404,Z 279.503,A -85,B 0,C 180,E1 -27277.999,E2 -27277.999} C_VEL
LIN {X 0,Y 91.78,Z 272.579,A -85,B 0,C 180,E1 -27284.412,E2 -27284.412} C_VEL
LIN {X 0,Y 95.357,Z 265.502,A -85,B 0,C 180,E1 -27289.371,E2 -27289.371} C_VEL
LIN {X 0,Y 99.52,Z 256.965,A -85,B 0,C 180,E1 -27293.959,E2 -27293.959} C_VEL
LIN {X 0,Y 104.179,Z 246.415,A -85,B 0,C 180,E1 -27298.18,E2 -27298.18} C_VEL
LIN {X 0,Y 108.545,Z 234.595,A -85,B 0,C 180,E1 -27301.742,E2 -27301.742} C_VEL
LIN {X 0,Y 112.307,Z 222.624,A -85,B 0,C 180,E1 -27304.279,E2 -27304.279} C_VEL
LIN {X 0,Y 115.38,Z 210.165,A -85,B 0,C 180,E1 -27306.164,E2 -27306.164} C_VEL
LIN {X 0,Y 117.611,Z 197.1,A -85,B 0,C 180,E1 -27307.524,E2 -27307.524} C_VEL
LIN {X 0,Y 119.129,Z 181.511,A -85,B 0,C 180,E1 -27308.444,E2 -27308.444} C_VEL
LIN {X 0,Y 121.364,Z 153.778,A -85,B 0,C 180,E1 -27309.72,E2 -27309.72} C_VEL
LIN {X 0,Y 117.675,Z 145.486,A -85,B 0,C 180,E1 -27312.516,E2 -27312.516} C_VEL
LIN {X 0,Y 114.257,Z 138.834,A -85,B 0,C 180,E1 -27315.331,E2 -27315.331} C_VEL
LIN {X 0,Y 109.943,Z 131.482,A -85,B 0,C 180,E1 -27319.334,E2 -27319.334} C_VEL
LIN {X 0,Y 106.606,Z 126.563,A -85,B 0,C 180,E1 -27322.899,E2 -27322.899} C_VEL
LIN {X 0,Y 104.272,Z 123.095,A -85,B 0,C 180,E1 -27325.792,E2 -27325.792} C_VEL
LIN {X 0,Y 101.79,Z 119.724,A -85,B 0,C 180,E1 -27329.343,E2 -27329.343} C_VEL
LIN {X 0,Y 101.173,Z 118.761,A -85,B 0,C 180,E1 -27330.363,E2 -27330.363} C_VEL
LIN {X 0,Y 98.853,Z 116.462,A -85,B 0,C 180,E1 -27334.502,E2 -27334.502} C_VEL
LIN {X 0,Y 97.551,Z 113.688,A -85,B 0,C 180,E1 -27337.829,E2 -27337.829} C_VEL
LIN {X 0,Y 94.733,Z 111.364,A -85,B 0,C 180,E1 -27350.39,E2 -27350.39} C_VEL
LIN {X 0,Y 95.24,Z 111.298,A -85,B 0,C 180,E1 -27358.942,E2 -27358.942} C_VEL
LIN {X 0,Y 97.516,Z 113.426,A -85,B 0,C 180,E1 -27367.245,E2 -27367.245} C_VEL
LIN {X 0,Y 98.036,Z 113.876,A -85,B 0,C 180,E1 -27368.502,E2 -27368.502} C_VEL
LIN {X 0,Y 99.642,Z 117.103,A -85,B 0,C 180,E1 -27372.215,E2 -27372.215} C_VEL
LIN {X 0,Y 101.823,Z 119.379,A -85,B 0,C 180,E1 -27375.863,E2 -27375.863} C_VEL
LIN {X 0,Y 104.166,Z 122.897,A -85,B 0,C 180,E1 -27379.298,E2 -27379.298} C_VEL
LIN {X 0,Y 105.296,Z 124.492,A -85,B 0,C 180,E1 -27380.75,E2 -27380.75} C_VEL
LIN {X 0,Y 108.464,Z 129.263,A -85,B 0,C 180,E1 -27384.39,E2 -27384.39} C_VEL
LIN {X 0,Y 111.861,Z 134.587,A -85,B 0,C 180,E1 -27387.746,E2 -27387.746} C_VEL
LIN {X 0,Y 114.982,Z 140.479,A -85,B 0,C 180,E1 -27390.548,E2 -27390.548} C_VEL
LIN {X 0,Y 118.777,Z 151.388,A -85,B 0,C 180,E1 -27393.897,E2 -27393.897} C_VEL
LIN {X 0,Y 120.013,Z 156.049,A -85,B 0,C 180,E1 -27394.996,E2 -27394.996} C_VEL
LIN {X 0,Y 120.215,Z 170.383,A -85,B 0,C 180,E1 -27396.364,E2 -27396.364} C_VEL
LIN {X 0,Y 117.507,Z 202.108,A -85,B 0,C 180,E1 -27397.899,E2 -27397.899} C_VEL
LIN {X 0,Y 115.438,Z 215.445,A -85,B 0,C 180,E1 -27399.081,E2 -27399.081} C_VEL
LIN {X 0,Y 112.371,Z 228.038,A -85,B 0,C 180,E1 -27400.681,E2 -27400.681} C_VEL
LIN {X 0,Y 108.928,Z 239.281,A -85,B 0,C 180,E1 -27402.783,E2 -27402.783} C_VEL
LIN {X 0,Y 104.488,Z 250.938,A -85,B 0,C 180,E1 -27405.745,E2 -27405.745} C_VEL
LIN {X 0,Y 99.969,Z 261.451,A -85,B 0,C 180,E1 -27409.435,E2 -27409.435} C_VEL
LIN {X 0,Y 95.347,Z 271.281,A -85,B 0,C 180,E1 -27414.174,E2 -27414.174} C_VEL
LIN {X 0,Y 92.348,Z 277.188,A -85,B 0,C 180,E1 -27417.809,E2 -27417.809} C_VEL
LIN {X 0,Y 88.716,Z 285.081,A -85,B 0,C 180,E1 -27424.168,E2 -27424.168} C_VEL
LIN {X 0,Y 85.998,Z 291.36,A -85,B 0,C 180,E1 -27430.918,E2 -27430.918} C_VEL
LIN {X 0,Y 84.525,Z 296.338,A -85,B 0,C 180,E1 -27438.001,E2 -27438.001} C_VEL
LIN {X 0,Y 84.284,Z 300.157,A -85,B 0,C 180,E1 -27445.215,E2 -27445.215} C_VEL
LIN {X 0,Y 84.464,Z 302.092,A -85,B 0,C 180,E1 -27449.998,E2 -27449.998} C_VEL
LIN {X 0,Y 84.271,Z 303.536,A -85,B 0,C 180,E1 -27454.782,E2 -27454.782} C_VEL
LIN {X 0,Y 84.982,Z 305.116,A -85,B 0,C 180,E1 -27464.363,E2 -27464.363} C_VEL
LIN {X 0,Y 87.877,Z 305.184,A -85,B 0,C 180,E1 -27473.568,E2 -27473.568} C_VEL
LIN {X 0,Y 90.252,Z 304.649,A -85,B 0,C 180,E1 -27477.853,E2 -27477.853} C_VEL
LIN {X 0,Y 96.404,Z 302.374,A -85,B 0,C 180,E1 -27485.675,E2 -27485.675} C_VEL
LIN {X 0,Y 101.122,Z 300.107,A -85,B 0,C 180,E1 -27490.138,E2 -27490.138} C_VEL
LIN {X 0,Y 108.415,Z 295.881,A -85,B 0,C 180,E1 -27495.483,E2 -27495.483} C_VEL
LIN {X 0,Y 115.572,Z 291.066,A -85,B 0,C 180,E1 -27499.474,E2 -27499.474} C_VEL
LIN {X 0,Y 124.642,Z 283.904,A -85,B 0,C 180,E1 -27503.463,E2 -27503.463} C_VEL
LIN {X 0,Y 132.769,Z 276.155,A -85,B 0,C 180,E1 -27506.48,E2 -27506.48} C_VEL
LIN {X 0,Y 139.909,Z 268.264,A -85,B 0,C 180,E1 -27508.642,E2 -27508.642} C_VEL
LIN {X 0,Y 147.302,Z 258.658,A -85,B 0,C 180,E1 -27510.542,E2 -27510.542} C_VEL
LIN {X 0,Y 154.15,Z 248.011,A -85,B 0,C 180,E1 -27512.046,E2 -27512.046} C_VEL
LIN {X 0,Y 159.542,Z 237.743,A -85,B 0,C 180,E1 -27513.128,E2 -27513.128} C_VEL
LIN {X 0,Y 164.601,Z 225.512,A -85,B 0,C 180,E1 -27514.074,E2 -27514.074} C_VEL
LIN {X 0,Y 168.475,Z 212.774,A -85,B 0,C 180,E1 -27514.785,E2 -27514.785} C_VEL
LIN {X 0,Y 170.876,Z 201.144,A -85,B 0,C 180,E1 -27515.252,E2 -27515.252} C_VEL
LIN {X 0,Y 170.719,Z 199.748,A -85,B 0,C 180,E1 -27515.691,E2 -27515.691} C_VEL
LIN {X 0,Y 168.977,Z 193.098,A -85,B 0,C 180,E1 -27518.819,E2 -27518.819} C_VEL
LIN {X 0,Y 168.768,Z 192.368,A -85,B 0,C 180,E1 -27519.214,E2 -27519.214} C_VEL
LIN {X 0,Y 168.208,Z 190.383,A -85,B 0,C 180,E1 -27520.343,E2 -27520.343} C_VEL
LIN {X 0,Y 167.212,Z 188.696,A -85,B 0,C 180,E1 -27522.246,E2 -27522.246} C_VEL
LIN {X 0,Y 166.218,Z 188.13,A -85,B 0,C 180,E1 -27524.26,E2 -27524.26} C_VEL
LIN {X 0,Y 164.342,Z 188.205,A -85,B 0,C 180,E1 -27529.985,E2 -27529.985} C_VEL
LIN {X 0,Y 164.13,Z 187.986,A -85,B 0,C 180,E1 -27535.088,E2 -27535.088} C_VEL
LIN {X 0,Y 164.466,Z 188.381,A -85,B 0,C 180,E1 -27537.551,E2 -27537.551} C_VEL
LIN {X 0,Y 165.715,Z 191.939,A -85,B 0,C 180,E1 -27542.583,E2 -27542.583} C_VEL
LIN {X 0,Y 167.068,Z 195.598,A -85,B 0,C 180,E1 -27546.037,E2 -27546.037} C_VEL
LIN {X 0,Y 168.522,Z 200.026,A -85,B 0,C 180,E1 -27549.225,E2 -27549.225} C_VEL
LIN {X 0,Y 165.493,Z 212.518,A -85,B 0,C 180,E1 -27549.927,E2 -27549.927} C_VEL
LIN {X 0,Y 161.029,Z 225.376,A -85,B 0,C 180,E1 -27550.895,E2 -27550.895} C_VEL
LIN {X 0,Y 156.27,Z 235.911,A -85,B 0,C 180,E1 -27551.998,E2 -27551.998} C_VEL
LIN {X 0,Y 149.982,Z 246.914,A -85,B 0,C 180,E1 -27553.476,E2 -27553.476} C_VEL
LIN {X 0,Y 142.959,Z 256.908,A -85,B 0,C 180,E1 -27555.256,E2 -27555.256} C_VEL
LIN {X 0,Y 134.612,Z 266.726,A -85,B 0,C 180,E1 -27557.675,E2 -27557.675} C_VEL
LIN {X 0,Y 125.797,Z 275.192,A -85,B 0,C 180,E1 -27560.649,E2 -27560.649} C_VEL
LIN {X 0,Y 117.351,Z 281.945,A -85,B 0,C 180,E1 -27564.038,E2 -27564.038} C_VEL
LIN {X 0,Y 110.708,Z 286.446,A -85,B 0,C 180,E1 -27567.287,E2 -27567.287} C_VEL
LIN {X 0,Y 103.216,Z 290.707,A -85,B 0,C 180,E1 -27571.669,E2 -27571.669} C_VEL
LIN {X 0,Y 96.381,Z 293.831,A -85,B 0,C 180,E1 -27576.671,E2 -27576.671} C_VEL
LIN {X 0,Y 92.262,Z 295.353,A -85,B 0,C 180,E1 -27580.384,E2 -27580.384} C_VEL
LIN {X 0,Y 86.554,Z 296.83,A -85,B 0,C 180,E1 -27586.954,E2 -27586.954} C_VEL
LIN {X 0,Y 82.53,Z 297.224,A -85,B 0,C 180,E1 -27593.412,E2 -27593.412} C_VEL
LIN {X 0,Y 80.326,Z 297.006,A -85,B 0,C 180,E1 -27598.337,E2 -27598.337} C_VEL
LIN {X 0,Y 78.637,Z 296.351,A -85,B 0,C 180,E1 -27603.46,E2 -27603.46} C_VEL
LIN {X 0,Y 77.481,Z 295.3,A -85,B 0,C 180,E1 -27608.728,E2 -27608.728} C_VEL
LIN {X 0,Y 76.855,Z 293.845,A -85,B 0,C 180,E1 -27614.08,E2 -27614.08} C_VEL
LIN {X 0,Y 77.117,Z 290.792,A -85,B 0,C 180,E1 -27622.145,E2 -27622.145} C_VEL
LIN {X 0,Y 78.478,Z 286.695,A -85,B 0,C 180,E1 -27630.002,E2 -27630.002} C_VEL
LIN {X 0,Y 81.342,Z 280.425,A -85,B 0,C 180,E1 -27638.698,E2 -27638.698} C_VEL
LIN {X 0,Y 84.903,Z 273.618,A -85,B 0,C 180,E1 -27645.608,E2 -27645.608} C_VEL
LIN {X 0,Y 89.487,Z 265.157,A -85,B 0,C 180,E1 -27651.906,E2 -27651.906} C_VEL
LIN {X 0,Y 94,Z 256.426,A -85,B 0,C 180,E1 -27656.655,E2 -27656.655} C_VEL
LIN {X 0,Y 99.034,Z 245.68,A -85,B 0,C 180,E1 -27660.966,E2 -27660.966} C_VEL
LIN {X 0,Y 103.127,Z 235.065,A -85,B 0,C 180,E1 -27664.212,E2 -27664.212} C_VEL
LIN {X 0,Y 107.091,Z 223.127,A -85,B 0,C 180,E1 -27666.789,E2 -27666.789} C_VEL
LIN {X 0,Y 110.338,Z 210.698,A -85,B 0,C 180,E1 -27668.684,E2 -27668.684} C_VEL
LIN {X 0,Y 112.628,Z 198.131,A -85,B 0,C 180,E1 -27670.025,E2 -27670.025} C_VEL
LIN {X 0,Y 114.086,Z 184.467,A -85,B 0,C 180,E1 -27670.889,E2 -27670.889} C_VEL
LIN {X 0,Y 116.474,Z 155.96,A -85,B 0,C 180,E1 -27672.222,E2 -27672.222} C_VEL
LIN {X 0,Y 112.158,Z 146.375,A -85,B 0,C 180,E1 -27675.968,E2 -27675.968} C_VEL
LIN {X 0,Y 107.707,Z 138.232,A -85,B 0,C 180,E1 -27680.37,E2 -27680.37} C_VEL
LIN {X 0,Y 104.372,Z 132.828,A -85,B 0,C 180,E1 -27684.235,E2 -27684.235} C_VEL
LIN {X 0,Y 102.154,Z 129.39,A -85,B 0,C 180,E1 -27687.224,E2 -27687.224} C_VEL
LIN {X 0,Y 99.725,Z 125.784,A -85,B 0,C 180,E1 -27691.091,E2 -27691.091} C_VEL
LIN {X 0,Y 96.869,Z 122.233,A -85,B 0,C 180,E1 -27696.903,E2 -27696.903} C_VEL
LIN {X 0,Y 96.119,Z 120.537,A -85,B 0,C 180,E1 -27699.142,E2 -27699.142} C_VEL
LIN {X 0,Y 93.817,Z 118.314,A -85,B 0,C 180,E1 -27711.382,E2 -27711.382} C_VEL
LIN {X 0,Y 94.434,Z 118.492,A -85,B 0,C 180,E1 -27719.466,E2 -27719.466} C_VEL
LIN {X 0,Y 96.607,Z 120.704,A -85,B 0,C 180,E1 -27727.313,E2 -27727.313} C_VEL
LIN {X 0,Y 98.18,Z 123.864,A -85,B 0,C 180,E1 -27731.254,E2 -27731.254} C_VEL
LIN {X 0,Y 100.042,Z 126.015,A -85,B 0,C 180,E1 -27734.642,E2 -27734.642} C_VEL
LIN {X 0,Y 102.348,Z 129.503,A -85,B 0,C 180,E1 -27738.257,E2 -27738.257} C_VEL
LIN {X 0,Y 105.966,Z 135.346,A -85,B 0,C 180,E1 -27742.929,E2 -27742.929} C_VEL
LIN {X 0,Y 109.311,Z 141.089,A -85,B 0,C 180,E1 -27746.539,E2 -27746.539} C_VEL
LIN {X 0,Y 111.385,Z 145.327,A -85,B 0,C 180,E1 -27748.596,E2 -27748.596} C_VEL
LIN {X 0,Y 114.538,Z 154.98,A -85,B 0,C 180,E1 -27751.733,E2 -27751.733} C_VEL
LIN {X 0,Y 115.385,Z 158.184,A -85,B 0,C 180,E1 -27752.571,E2 -27752.571} C_VEL
LIN {X 0,Y 115.47,Z 170.218,A -85,B 0,C 180,E1 -27753.781,E2 -27753.781} C_VEL
LIN {X 0,Y 112.591,Z 202.303,A -85,B 0,C 180,E1 -27755.365,E2 -27755.365} C_VEL
LIN {X 0,Y 110.267,Z 216.107,A -85,B 0,C 180,E1 -27756.611,E2 -27756.611} C_VEL
LIN {X 0,Y 106.937,Z 228.882,A -85,B 0,C 180,E1 -27758.32,E2 -27758.32} C_VEL
LIN {X 0,Y 103.05,Z 240.659,A -85,B 0,C 180,E1 -27760.646,E2 -27760.646} C_VEL
LIN {X 0,Y 98.341,Z 251.972,A -85,B 0,C 180,E1 -27763.646,E2 -27763.646} C_VEL
LIN {X 0,Y 94.136,Z 261.168,A -85,B 0,C 180,E1 -27767.056,E2 -27767.056} C_VEL
LIN {X 0,Y 89.183,Z 270.999,A -85,B 0,C 180,E1 -27772.002,E2 -27772.002} C_VEL
LIN {X 0,Y 86.327,Z 276.112,A -85,B 0,C 180,E1 -27775.256,E2 -27775.256} C_VEL
LIN {X 0,Y 82.308,Z 284.173,A -85,B 0,C 180,E1 -27781.988,E2 -27781.988} C_VEL
LIN {X 0,Y 79.259,Z 290.557,A -85,B 0,C 180,E1 -27789.224,E2 -27789.224} C_VEL
LIN {X 0,Y 77.56,Z 295.626,A -85,B 0,C 180,E1 -27796.905,E2 -27796.905} C_VEL
LIN {X 0,Y 77.195,Z 299.53,A -85,B 0,C 180,E1 -27804.775,E2 -27804.775} C_VEL
LIN {X 0,Y 77.395,Z 301.508,A -85,B 0,C 180,E1 -27809.998,E2 -27809.998} C_VEL
LIN {X 0,Y 77.187,Z 302.989,A -85,B 0,C 180,E1 -27815.222,E2 -27815.222} C_VEL
LIN {X 0,Y 77.343,Z 304.043,A -85,B 0,C 180,E1 -27820.469,E2 -27820.469} C_VEL
LIN {X 0,Y 79.458,Z 304.932,A -85,B 0,C 180,E1 -27830.718,E2 -27830.718} C_VEL
LIN {X 0,Y 84.017,Z 304.335,A -85,B 0,C 180,E1 -27840.124,E2 -27840.124} C_VEL
LIN {X 0,Y 90.702,Z 302.152,A -85,B 0,C 180,E1 -27848.305,E2 -27848.305} C_VEL
LIN {X 0,Y 95.241,Z 300.198,A -85,B 0,C 180,E1 -27852.446,E2 -27852.446} C_VEL
LIN {X 0,Y 103.56,Z 295.818,A -85,B 0,C 180,E1 -27858.286,E2 -27858.286} C_VEL
LIN {X 0,Y 111.082,Z 291.09,A -85,B 0,C 180,E1 -27862.263,E2 -27862.263} C_VEL
LIN {X 0,Y 120.562,Z 284.023,A -85,B 0,C 180,E1 -27866.167,E2 -27866.167} C_VEL
LIN {X 0,Y 128.989,Z 276.42,A -85,B 0,C 180,E1 -27869.107,E2 -27869.107} C_VEL
LIN {X 0,Y 136.361,Z 268.671,A -85,B 0,C 180,E1 -27871.182,E2 -27871.182} C_VEL
LIN {X 0,Y 143.954,Z 259.24,A -85,B 0,C 180,E1 -27872.995,E2 -27872.995} C_VEL
LIN {X 0,Y 150.966,Z 248.793,A -85,B 0,C 180,E1 -27874.417,E2 -27874.417} C_VEL
LIN {X 0,Y 157.276,Z 237.207,A -85,B 0,C 180,E1 -27875.568,E2 -27875.568} C_VEL
LIN {X 0,Y 162.453,Z 224.865,A -85,B 0,C 180,E1 -27876.461,E2 -27876.461} C_VEL
LIN {X 0,Y 166.334,Z 212.349,A -85,B 0,C 180,E1 -27877.106,E2 -27877.106} C_VEL
LIN {X 0,Y 168.146,Z 204.086,A -85,B 0,C 180,E1 -27877.497,E2 -27877.497} C_VEL
LIN {X 0,Y 166.971,Z 198.001,A -85,B 0,C 180,E1 -27880.563,E2 -27880.563} C_VEL
LIN {X 0,Y 165.851,Z 193.682,A -85,B 0,C 180,E1 -27883.538,E2 -27883.538} C_VEL
LIN {X 0,Y 165.168,Z 191.032,A -85,B 0,C 180,E1 -27885.838,E2 -27885.838} C_VEL
LIN {X 0,Y 164.342,Z 188.205,A -85,B 0,C 180,E1 -27889.985,E2 -27889.985} C_VEL
LIN {X 0,Y 164.039,Z 188.598,A -85,B 0,C 180,E1 -27892.041,E2 -27892.041} C_VEL
LIN {X 0,Y 163.798,Z 190.178,A -85,B 0,C 180,E1 -27894.048,E2 -27894.048} C_VEL
LIN {X 0,Y 163.735,Z 196.402,A -85,B 0,C 180,E1 -27899.286,E2 -27899.286} C_VEL
LIN {X 0,Y 163.939,Z 197.631,A -85,B 0,C 180,E1 -27900.639,E2 -27900.639} C_VEL
LIN {X 0,Y 164.419,Z 199.316,A -85,B 0,C 180,E1 -27902.604,E2 -27902.604} C_VEL
LIN {X 0,Y 165.404,Z 202.773,A -85,B 0,C 180,E1 -27905.869,E2 -27905.869} C_VEL
LIN {X 0,Y 165.791,Z 204.443,A -85,B 0,C 180,E1 -27907.077,E2 -27907.077} C_VEL
LIN {X 0,Y 162.411,Z 216.603,A -85,B 0,C 180,E1 -27907.799,E2 -27907.799} C_VEL
LIN {X 0,Y 157.895,Z 228.249,A -85,B 0,C 180,E1 -27908.675,E2 -27908.675} C_VEL
LIN {X 0,Y 152.456,Z 239.236,A -85,B 0,C 180,E1 -27909.825,E2 -27909.825} C_VEL
LIN {X 0,Y 145.988,Z 249.732,A -85,B 0,C 180,E1 -27911.257,E2 -27911.257} C_VEL
LIN {X 0,Y 138.823,Z 259.242,A -85,B 0,C 180,E1 -27912.962,E2 -27912.962} C_VEL
LIN {X 0,Y 131.012,Z 267.837,A -85,B 0,C 180,E1 -27915.079,E2 -27915.079} C_VEL
LIN {X 0,Y 121.891,Z 276.173,A -85,B 0,C 180,E1 -27917.948,E2 -27917.948} C_VEL
LIN {X 0,Y 113.104,Z 282.814,A -85,B 0,C 180,E1 -27921.246,E2 -27921.246} C_VEL
LIN {X 0,Y 104.796,Z 288.01,A -85,B 0,C 180,E1 -27925.133,E2 -27925.133} C_VEL
LIN {X 0,Y 96.993,Z 291.976,A -85,B 0,C 180,E1 -27929.602,E2 -27929.602} C_VEL
LIN {X 0,Y 92.139,Z 293.985,A -85,B 0,C 180,E1 -27932.965,E2 -27932.965} C_VEL
LIN {X 0,Y 87.641,Z 295.556,A -85,B 0,C 180,E1 -27936.69,E2 -27936.69} C_VEL
LIN {X 0,Y 80.689,Z 297.24,A -85,B 0,C 180,E1 -27944.173,E2 -27944.173} C_VEL
LIN {X 0,Y 76.721,Z 297.601,A -85,B 0,C 180,E1 -27950.119,E2 -27950.119} C_VEL
LIN {X 0,Y 74.155,Z 297.455,A -85,B 0,C 180,E1 -27955.346,E2 -27955.346} C_VEL
LIN {X 0,Y 71.872,Z 296.734,A -85,B 0,C 180,E1 -27961.653,E2 -27961.653} C_VEL
LIN {X 0,Y 69.863,Z 294.442,A -85,B 0,C 180,E1 -27972.437,E2 -27972.437} C_VEL
LIN {X 0,Y 69.944,Z 291.474,A -85,B 0,C 180,E1 -27981.333,E2 -27981.333} C_VEL
LIN {X 0,Y 71.294,Z 287.47,A -85,B 0,C 180,E1 -27990.002,E2 -27990.002} C_VEL
LIN {X 0,Y 73.744,Z 282.342,A -85,B 0,C 180,E1 -27998.221,E2 -27998.221} C_VEL
LIN {X 0,Y 77.352,Z 275.902,A -85,B 0,C 180,E1 -28005.819,E2 -28005.819} C_VEL
LIN {X 0,Y 82.055,Z 267.851,A -85,B 0,C 180,E1 -28012.672,E2 -28012.672} C_VEL
LIN {X 0,Y 86.712,Z 259.644,A -85,B 0,C 180,E1 -28017.779,E2 -28017.779} C_VEL
LIN {X 0,Y 91.845,Z 249.654,A -85,B 0,C 180,E1 -28022.389,E2 -28022.389} C_VEL
LIN {X 0,Y 96.243,Z 239.801,A -85,B 0,C 180,E1 -28025.747,E2 -28025.747} C_VEL
LIN {X 0,Y 100.263,Z 229.116,A -85,B 0,C 180,E1 -28028.471,E2 -28028.471} C_VEL
LIN {X 0,Y 104.307,Z 216.192,A -85,B 0,C 180,E1 -28030.749,E2 -28030.749} C_VEL
LIN {X 0,Y 107.139,Z 203.496,A -85,B 0,C 180,E1 -28032.339,E2 -28032.339} C_VEL
LIN {X 0,Y 109.025,Z 190.012,A -85,B 0,C 180,E1 -28033.396,E2 -28033.396} C_VEL
LIN {X 0,Y 111.852,Z 158.57,A -85,B 0,C 180,E1 -28034.874,E2 -28034.874} C_VEL
LIN {X 0,Y 108.145,Z 150.044,A -85,B 0,C 180,E1 -28038.554,E2 -28038.554} C_VEL
LIN {X 0,Y 104.443,Z 142.96,A -85,B 0,C 180,E1 -28042.726,E2 -28042.726} C_VEL
LIN {X 0,Y 101.278,Z 137.687,A -85,B 0,C 180,E1 -28046.905,E2 -28046.905} C_VEL
LIN {X 0,Y 99.997,Z 135.586,A -85,B 0,C 180,E1 -28048.871,E2 -28048.871} C_VEL
LIN {X 0,Y 97.724,Z 131.961,A -85,B 0,C 180,E1 -28052.927,E2 -28052.927} C_VEL
LIN {X 0,Y 95.456,Z 128.901,A -85,B 0,C 180,E1 -28058.135,E2 -28058.135} C_VEL
LIN {X 0,Y 94.815,Z 127.404,A -85,B 0,C 180,E1 -28060.271,E2 -28060.271} C_VEL
LIN {X 0,Y 92.941,Z 125.372,A -85,B 0,C 180,E1 -28071.3,E2 -28071.3} C_VEL
LIN {X 0,Y 93.455,Z 125.483,A -85,B 0,C 180,E1 -28078.922,E2 -28078.922} C_VEL
LIN {X 0,Y 95.227,Z 127.476,A -85,B 0,C 180,E1 -28086.089,E2 -28086.089} C_VEL
LIN {X 0,Y 96.95,Z 130.876,A -85,B 0,C 180,E1 -28090.704,E2 -28090.704} C_VEL
LIN {X 0,Y 98.204,Z 132.487,A -85,B 0,C 180,E1 -28093.183,E2 -28093.183} C_VEL
LIN {X 0,Y 100.85,Z 136.79,A -85,B 0,C 180,E1 -28097.652,E2 -28097.652} C_VEL
LIN {X 0,Y 104.585,Z 143.179,A -85,B 0,C 180,E1 -28102.684,E2 -28102.684} C_VEL
LIN {X 0,Y 107.73,Z 149.445,A -85,B 0,C 180,E1 -28106.271,E2 -28106.271} C_VEL
LIN {X 0,Y 110.658,Z 159.322,A -85,B 0,C 180,E1 -28109.616,E2 -28109.616} C_VEL
LIN {X 0,Y 110.966,Z 161.349,A -85,B 0,C 180,E1 -28110.048,E2 -28110.048} C_VEL
LIN {X 0,Y 110.833,Z 171.893,A -85,B 0,C 180,E1 -28111.078,E2 -28111.078} C_VEL
LIN {X 0,Y 107.968,Z 202.122,A -85,B 0,C 180,E1 -28112.578,E2 -28112.578} C_VEL
LIN {X 0,Y 105.492,Z 216.005,A -85,B 0,C 180,E1 -28113.828,E2 -28113.828} C_VEL
LIN {X 0,Y 102.01,Z 228.685,A -85,B 0,C 180,E1 -28115.526,E2 -28115.526} C_VEL
LIN {X 0,Y 97.917,Z 240.424,A -85,B 0,C 180,E1 -28117.857,E2 -28117.857} C_VEL
LIN {X 0,Y 92.97,Z 251.714,A -85,B 0,C 180,E1 -28120.89,E2 -28120.89} C_VEL
LIN {X 0,Y 88.485,Z 260.885,A -85,B 0,C 180,E1 -28124.369,E2 -28124.369} C_VEL
LIN {X 0,Y 83.229,Z 270.629,A -85,B 0,C 180,E1 -28129.461,E2 -28129.461} C_VEL
LIN {X 0,Y 79.713,Z 276.557,A -85,B 0,C 180,E1 -28133.476,E2 -28133.476} C_VEL
LIN {X 0,Y 75.418,Z 284.418,A -85,B 0,C 180,E1 -28140.707,E2 -28140.707} C_VEL
LIN {X 0,Y 71.786,Z 291.596,A -85,B 0,C 180,E1 -28149.959,E2 -28149.959} C_VEL
LIN {X 0,Y 70.286,Z 296.361,A -85,B 0,C 180,E1 -28158.462,E2 -28158.462} C_VEL
LIN {X 0,Y 70.087,Z 298.9,A -85,B 0,C 180,E1 -28164.243,E2 -28164.243} C_VEL
LIN {X 0,Y 70.296,Z 301.31,A -85,B 0,C 180,E1 -28171.286,E2 -28171.286} C_VEL
LIN {X 0,Y 70.36,Z 303.545,A -85,B 0,C 180,E1 -28181.522,E2 -28181.522} C_VEL
LIN {X 0,Y 71.276,Z 304.234,A -85,B 0,C 180,E1 -28187.204,E2 -28187.204} C_VEL
LIN {X 0,Y 75.023,Z 304.447,A -85,B 0,C 180,E1 -28197.928,E2 -28197.928} C_VEL
LIN {X 0,Y 81.326,Z 303.178,A -85,B 0,C 180,E1 -28207.221,E2 -28207.221} C_VEL
LIN {X 0,Y 89.449,Z 300.284,A -85,B 0,C 180,E1 -28214.999,E2 -28214.999} C_VEL
LIN {X 0,Y 96.474,Z 297.036,A -85,B 0,C 180,E1 -28219.896,E2 -28219.896} C_VEL
LIN {X 0,Y 104.194,Z 292.76,A -85,B 0,C 180,E1 -28224.036,E2 -28224.036} C_VEL
LIN {X 0,Y 113.885,Z 286.324,A -85,B 0,C 180,E1 -28228.049,E2 -28228.049} C_VEL
LIN {X 0,Y 122.576,Z 279.349,A -85,B 0,C 180,E1 -28230.968,E2 -28230.968} C_VEL
LIN {X 0,Y 128.537,Z 273.752,A -85,B 0,C 180,E1 -28232.683,E2 -28232.683} C_VEL
LIN {X 0,Y 136.242,Z 265.537,A -85,B 0,C 180,E1 -28234.517,E2 -28234.517} C_VEL
LIN {X 0,Y 143.256,Z 256.63,A -85,B 0,C 180,E1 -28236.023,E2 -28236.023} C_VEL
LIN {X 0,Y 150.451,Z 245.695,A -85,B 0,C 180,E1 -28237.304,E2 -28237.304} C_VEL
LIN {X 0,Y 156.924,Z 233.244,A -85,B 0,C 180,E1 -28238.325,E2 -28238.325} C_VEL
LIN {X 0,Y 161.666,Z 221.321,A -85,B 0,C 180,E1 -28239.076,E2 -28239.076} C_VEL
LIN {X 0,Y 165.405,Z 208.337,A -85,B 0,C 180,E1 -28239.62,E2 -28239.62} C_VEL
LIN {X 0,Y 165.484,Z 207.436,A -85,B 0,C 180,E1 -28239.818,E2 -28239.818} C_VEL
LIN {X 0,Y 164.828,Z 202.872,A -85,B 0,C 180,E1 -28242.475,E2 -28242.475} C_VEL
LIN {X 0,Y 164.262,Z 199.664,A -85,B 0,C 180,E1 -28244.808,E2 -28244.808} C_VEL
LIN {X 0,Y 163.969,Z 197.867,A -85,B 0,C 180,E1 -28246.365,E2 -28246.365} C_VEL
LIN {X 0,Y 163.345,Z 195.276,A -85,B 0,C 180,E1 -28250.168,E2 -28250.168} C_VEL
LIN {X 0,Y 163.157,Z 195.007,A -85,B 0,C 180,E1 -28255.058,E2 -28255.058} C_VEL
LIN {X 0,Y 163.408,Z 195.406,A -85,B 0,C 180,E1 -28257.227,E2 -28257.227} C_VEL
LIN {X 0,Y 163.939,Z 197.631,A -85,B 0,C 180,E1 -28260.639,E2 -28260.639} C_VEL
LIN {X 0,Y 164.126,Z 199.349,A -85,B 0,C 180,E1 -28261.942,E2 -28261.942} C_VEL
LIN {X 0,Y 164.032,Z 202.035,A -85,B 0,C 180,E1 -28263.048,E2 -28263.048} C_VEL
LIN {X 0,Y 163.471,Z 206.557,A -85,B 0,C 180,E1 -28264.202,E2 -28264.202} C_VEL
LIN {X 0,Y 162.274,Z 212.027,A -85,B 0,C 180,E1 -28265.022,E2 -28265.022} C_VEL
LIN {X 0,Y 161.56,Z 214.372,A -85,B 0,C 180,E1 -28265.198,E2 -28265.198} C_VEL
LIN {X 0,Y 157.091,Z 226.439,A -85,B 0,C 180,E1 -28265.996,E2 -28265.996} C_VEL
LIN {X 0,Y 151.378,Z 238.146,A -85,B 0,C 180,E1 -28267.089,E2 -28267.089} C_VEL
LIN {X 0,Y 144.97,Z 248.564,A -85,B 0,C 180,E1 -28268.363,E2 -28268.363} C_VEL
LIN {X 0,Y 137.363,Z 258.639,A -85,B 0,C 180,E1 -28269.975,E2 -28269.975} C_VEL
LIN {X 0,Y 129.292,Z 267.455,A -85,B 0,C 180,E1 -28271.926,E2 -28271.926} C_VEL
LIN {X 0,Y 119.823,Z 275.921,A -85,B 0,C 180,E1 -28274.59,E2 -28274.59} C_VEL
LIN {X 0,Y 110.65,Z 282.677,A -85,B 0,C 180,E1 -28277.692,E2 -28277.692} C_VEL
LIN {X 0,Y 101.872,Z 287.999,A -85,B 0,C 180,E1 -28281.359,E2 -28281.359} C_VEL
LIN {X 0,Y 93.563,Z 292.071,A -85,B 0,C 180,E1 -28285.664,E2 -28285.664} C_VEL
LIN {X 0,Y 88.329,Z 294.139,A -85,B 0,C 180,E1 -28288.932,E2 -28288.932} C_VEL
LIN {X 0,Y 83.423,Z 295.757,A -85,B 0,C 180,E1 -28292.603,E2 -28292.603} C_VEL
LIN {X 0,Y 78.909,Z 296.949,A -85,B 0,C 180,E1 -28296.722,E2 -28296.722} C_VEL
LIN {X 0,Y 74.793,Z 297.676,A -85,B 0,C 180,E1 -28301.263,E2 -28301.263} C_VEL
LIN {X 0,Y 71.208,Z 297.979,A -85,B 0,C 180,E1 -28306.303,E2 -28306.303} C_VEL
LIN {X 0,Y 68.203,Z 297.879,A -85,B 0,C 180,E1 -28311.812,E2 -28311.812} C_VEL
LIN {X 0,Y 65.225,Z 297.105,A -85,B 0,C 180,E1 -28319.545,E2 -28319.545} C_VEL
LIN {X 0,Y 62.933,Z 295.035,A -85,B 0,C 180,E1 -28330.429,E2 -28330.429} C_VEL
LIN {X 0,Y 62.757,Z 292.157,A -85,B 0,C 180,E1 -28340.332,E2 -28340.332} C_VEL
LIN {X 0,Y 64.106,Z 288.241,A -85,B 0,C 180,E1 -28350.002,E2 -28350.002} C_VEL
LIN {X 0,Y 66.677,Z 283.211,A -85,B 0,C 180,E1 -28359.099,E2 -28359.099} C_VEL
LIN {X 0,Y 70.522,Z 276.907,A -85,B 0,C 180,E1 -28367.398,E2 -28367.398} C_VEL
LIN {X 0,Y 75.517,Z 269.029,A -85,B 0,C 180,E1 -28374.76,E2 -28374.76} C_VEL
LIN {X 0,Y 81.542,Z 259.181,A -85,B 0,C 180,E1 -28381.142,E2 -28381.142} C_VEL
LIN {X 0,Y 87.081,Z 248.96,A -85,B 0,C 180,E1 -28385.814,E2 -28385.814} C_VEL
LIN {X 0,Y 91.769,Z 238.848,A -85,B 0,C 180,E1 -28389.186,E2 -28389.186} C_VEL
LIN {X 0,Y 96.076,Z 227.836,A -85,B 0,C 180,E1 -28391.876,E2 -28391.876} C_VEL
LIN {X 0,Y 100.016,Z 215.583,A -85,B 0,C 180,E1 -28393.942,E2 -28393.942} C_VEL
LIN {X 0,Y 102.933,Z 202.689,A -85,B 0,C 180,E1 -28395.469,E2 -28395.469} C_VEL
LIN {X 0,Y 104.883,Z 188.879,A -85,B 0,C 180,E1 -28396.484,E2 -28396.484} C_VEL
LIN {X 0,Y 107.46,Z 161.238,A -85,B 0,C 180,E1 -28397.764,E2 -28397.764} C_VEL
LIN {X 0,Y 104.638,Z 154.477,A -85,B 0,C 180,E1 -28400.984,E2 -28400.984} C_VEL
LIN {X 0,Y 101.714,Z 148.504,A -85,B 0,C 180,E1 -28404.708,E2 -28404.708} C_VEL
LIN {X 0,Y 98.294,Z 142.219,A -85,B 0,C 180,E1 -28409.966,E2 -28409.966} C_VEL
LIN {X 0,Y 95.818,Z 138.268,A -85,B 0,C 180,E1 -28414.825,E2 -28414.825} C_VEL
LIN {X 0,Y 93.867,Z 134.965,A -85,B 0,C 180,E1 -28420.221,E2 -28420.221} C_VEL
LIN {X 0,Y 93.599,Z 134.295,A -85,B 0,C 180,E1 -28421.267,E2 -28421.267} C_VEL
LIN {X 0,Y 92.063,Z 132.442,A -85,B 0,C 180,E1 -28431.217,E2 -28431.217} C_VEL
LIN {X 0,Y 92.485,Z 132.475,A -85,B 0,C 180,E1 -28438.366,E2 -28438.366} C_VEL
LIN {X 0,Y 93.949,Z 134.404,A -85,B 0,C 180,E1 -28445.045,E2 -28445.045} C_VEL
LIN {X 0,Y 95.902,Z 138.118,A -85,B 0,C 180,E1 -28450.522,E2 -28450.522} C_VEL
LIN {X 0,Y 96.804,Z 139.651,A -85,B 0,C 180,E1 -28452.462,E2 -28452.462} C_VEL
LIN {X 0,Y 99.02,Z 143.538,A -85,B 0,C 180,E1 -28456.492,E2 -28456.492} C_VEL
LIN {X 0,Y 101.909,Z 148.815,A -85,B 0,C 180,E1 -28460.784,E2 -28460.784} C_VEL
LIN {X 0,Y 104.449,Z 154.313,A -85,B 0,C 180,E1 -28464.06,E2 -28464.06} C_VEL
LIN {X 0,Y 106.787,Z 162.919,A -85,B 0,C 180,E1 -28467.138,E2 -28467.138} C_VEL
LIN {X 0,Y 106.563,Z 172.524,A -85,B 0,C 180,E1 -28468.1,E2 -28468.1} C_VEL
LIN {X 0,Y 103.651,Z 201.553,A -85,B 0,C 180,E1 -28469.501,E2 -28469.501} C_VEL
LIN {X 0,Y 101.156,Z 215.178,A -85,B 0,C 180,E1 -28470.718,E2 -28470.718} C_VEL
LIN {X 0,Y 97.665,Z 227.47,A -85,B 0,C 180,E1 -28472.269,E2 -28472.269} C_VEL
LIN {X 0,Y 93.047,Z 240.191,A -85,B 0,C 180,E1 -28474.772,E2 -28474.772} C_VEL
LIN {X 0,Y 87.828,Z 251.451,A -85,B 0,C 180,E1 -28477.794,E2 -28477.794} C_VEL
LIN {X 0,Y 83.057,Z 260.6,A -85,B 0,C 180,E1 -28481.323,E2 -28481.323} C_VEL
LIN {X 0,Y 77.333,Z 270.432,A -85,B 0,C 180,E1 -28486.637,E2 -28486.637} C_VEL
LIN {X 0,Y 73.199,Z 276.971,A -85,B 0,C 180,E1 -28491.383,E2 -28491.383} C_VEL
LIN {X 0,Y 68.58,Z 284.658,A -85,B 0,C 180,E1 -28499.174,E2 -28499.174} C_VEL
LIN {X 0,Y 65.114,Z 290.795,A -85,B 0,C 180,E1 -28507.802,E2 -28507.802} C_VEL
LIN {X 0,Y 63.298,Z 295.649,A -85,B 0,C 180,E1 -28517.168,E2 -28517.168} C_VEL
LIN {X 0,Y 63.03,Z 299.342,A -85,B 0,C 180,E1 -28526.802,E2 -28526.802} C_VEL
LIN {X 0,Y 63.251,Z 300.337,A -85,B 0,C 180,E1 -28529.998,E2 -28529.998} C_VEL
LIN {X 0,Y 63.046,Z 301.888,A -85,B 0,C 180,E1 -28536.398,E2 -28536.398} C_VEL
LIN {X 0,Y 64.491,Z 303.785,A -85,B 0,C 180,E1 -28549.08,E2 -28549.08} C_VEL
LIN {X 0,Y 68.811,Z 304.078,A -85,B 0,C 180,E1 -28560.706,E2 -28560.706} C_VEL
LIN {X 0,Y 75.775,Z 302.89,A -85,B 0,C 180,E1 -28570.482,E2 -28570.482} C_VEL
LIN {X 0,Y 83.859,Z 300.37,A -85,B 0,C 180,E1 -28577.899,E2 -28577.899} C_VEL
LIN {X 0,Y 92.04,Z 296.931,A -85,B 0,C 180,E1 -28583.295,E2 -28583.295} C_VEL
LIN {X 0,Y 100.177,Z 292.741,A -85,B 0,C 180,E1 -28587.335,E2 -28587.335} C_VEL
LIN {X 0,Y 110.298,Z 286.405,A -85,B 0,C 180,E1 -28591.176,E2 -28591.176} C_VEL
LIN {X 0,Y 119.291,Z 279.55,A -85,B 0,C 180,E1 -28593.952,E2 -28593.952} C_VEL
LIN {X 0,Y 125.447,Z 274.072,A -85,B 0,C 180,E1 -28595.555,E2 -28595.555} C_VEL
LIN {X 0,Y 133.344,Z 266.005,A -85,B 0,C 180,E1 -28597.269,E2 -28597.269} C_VEL
LIN {X 0,Y 141.35,Z 256.197,A -85,B 0,C 180,E1 -28598.786,E2 -28598.786} C_VEL
LIN {X 0,Y 148.693,Z 245.248,A -85,B 0,C 180,E1 -28599.947,E2 -28599.947} C_VEL
LIN {X 0,Y 155.284,Z 232.784,A -85,B 0,C 180,E1 -28600.868,E2 -28600.868} C_VEL
LIN {X 0,Y 159.96,Z 221.245,A -85,B 0,C 180,E1 -28601.539,E2 -28601.539} C_VEL
LIN {X 0,Y 162.97,Z 211.406,A -85,B 0,C 180,E1 -28601.978,E2 -28601.978} C_VEL
LIN {X 0,Y 162.526,Z 206.23,A -85,B 0,C 180,E1 -28605.523,E2 -28605.523} C_VEL
LIN {X 0,Y 162.327,Z 204.476,A -85,B 0,C 180,E1 -28607.181,E2 -28607.181} C_VEL
LIN {X 0,Y 162.01,Z 202.152,A -85,B 0,C 180,E1 -28610.638,E2 -28610.638} C_VEL
LIN {X 0,Y 161.852,Z 201.961,A -85,B 0,C 180,E1 -28615.018,E2 -28615.018} C_VEL
LIN {X 0,Y 161.989,Z 202.397,A -85,B 0,C 180,E1 -28617.001,E2 -28617.001} C_VEL
LIN {X 0,Y 162.466,Z 205.24,A -85,B 0,C 180,E1 -28621.24,E2 -28621.24} C_VEL
LIN {X 0,Y 163.149,Z 208.875,A -85,B 0,C 180,E1 -28624.866,E2 -28624.866} C_VEL
LIN {X 0,Y 161.56,Z 214.372,A -85,B 0,C 180,E1 -28625.198,E2 -28625.198} C_VEL
LIN {X 0,Y 159.549,Z 219.946,A -85,B 0,C 180,E1 -28625.31,E2 -28625.31} C_VEL
LIN {X 0,Y 155.333,Z 228.846,A -85,B 0,C 180,E1 -28624.915,E2 -28624.915} C_VEL
LIN {X 0,Y 150.494,Z 237.492,A -85,B 0,C 180,E1 -28624.591,E2 -28624.591} C_VEL
LIN {X 0,Y 147.491,Z 242.457,A -85,B 0,C 180,E1 -28624.849,E2 -28624.849} C_VEL
LIN {X 0,Y 140.476,Z 252.744,A -85,B 0,C 180,E1 -28626.108,E2 -28626.108} C_VEL
LIN {X 0,Y 132.942,Z 261.836,A -85,B 0,C 180,E1 -28627.608,E2 -28627.608} C_VEL
LIN {X 0,Y 125.045,Z 269.791,A -85,B 0,C 180,E1 -28629.389,E2 -28629.389} C_VEL
LIN {X 0,Y 116.575,Z 276.934,A -85,B 0,C 180,E1 -28631.58,E2 -28631.58} C_VEL
LIN {X 0,Y 108.623,Z 282.547,A -85,B 0,C 180,E1 -28633.956,E2 -28633.956} C_VEL
LIN {X 0,Y 99.414,Z 287.976,A -85,B 0,C 180,E1 -28637.381,E2 -28637.381} C_VEL
LIN {X 0,Y 90.6,Z 292.149,A -85,B 0,C 180,E1 -28641.436,E2 -28641.436} C_VEL
LIN {X 0,Y 84.999,Z 294.303,A -85,B 0,C 180,E1 -28644.566,E2 -28644.566} C_VEL
LIN {X 0,Y 79.677,Z 295.964,A -85,B 0,C 180,E1 -28648.112,E2 -28648.112} C_VEL
LIN {X 0,Y 74.723,Z 297.198,A -85,B 0,C 180,E1 -28652.173,E2 -28652.173} C_VEL
LIN {X 0,Y 69.642,Z 298.061,A -85,B 0,C 180,E1 -28657.267,E2 -28657.267} C_VEL
LIN {X 0,Y 62.562,Z 298.3,A -85,B 0,C 180,E1 -28667.625,E2 -28667.625} C_VEL
LIN {X 0,Y 58.644,Z 297.469,A -85,B 0,C 180,E1 -28677.027,E2 -28677.027} C_VEL
LIN {X 0,Y 56.106,Z 295.628,A -85,B 0,C 180,E1 -28687.93,E2 -28687.93} C_VEL
LIN {X 0,Y 55.572,Z 292.841,A -85,B 0,C 180,E1 -28699.067,E2 -28699.067} C_VEL
LIN {X 0,Y 56.878,Z 289.015,A -85,B 0,C 180,E1 -28710.003,E2 -28710.003} C_VEL
LIN {X 0,Y 59.616,Z 284.082,A -85,B 0,C 180,E1 -28720.188,E2 -28720.188} C_VEL
LIN {X 0,Y 63.729,Z 277.89,A -85,B 0,C 180,E1 -28729.322,E2 -28729.322} C_VEL
LIN {X 0,Y 69.105,Z 270.198,A -85,B 0,C 180,E1 -28737.238,E2 -28737.238} C_VEL
LIN {X 0,Y 74.414,Z 262.306,A -85,B 0,C 180,E1 -28742.894,E2 -28742.894} C_VEL
LIN {X 0,Y 80.22,Z 252.688,A -85,B 0,C 180,E1 -28747.828,E2 -28747.828} C_VEL
LIN {X 0,Y 85.173,Z 243.32,A -85,B 0,C 180,E1 -28751.311,E2 -28751.311} C_VEL
LIN {X 0,Y 90.25,Z 231.776,A -85,B 0,C 180,E1 -28754.498,E2 -28754.498} C_VEL
LIN {X 0,Y 94.725,Z 219.468,A -85,B 0,C 180,E1 -28756.723,E2 -28756.723} C_VEL
LIN {X 0,Y 98.137,Z 206.502,A -85,B 0,C 180,E1 -28758.4,E2 -28758.4} C_VEL
LIN {X 0,Y 100.404,Z 193.531,A -85,B 0,C 180,E1 -28759.499,E2 -28759.499} C_VEL
LIN {X 0,Y 103.35,Z 163.942,A -85,B 0,C 180,E1 -28760.9,E2 -28760.9} C_VEL
LIN {X 0,Y 100.965,Z 158.045,A -85,B 0,C 180,E1 -28764.073,E2 -28764.073} C_VEL
LIN {X 0,Y 98.53,Z 152.908,A -85,B 0,C 180,E1 -28767.707,E2 -28767.707} C_VEL
LIN {X 0,Y 96.055,Z 148.064,A -85,B 0,C 180,E1 -28772.158,E2 -28772.158} C_VEL
LIN {X 0,Y 94.356,Z 144.968,A -85,B 0,C 180,E1 -28775.979,E2 -28775.979} C_VEL
LIN {X 0,Y 92.531,Z 141.479,A -85,B 0,C 180,E1 -28781.758,E2 -28781.758} C_VEL
LIN {X 0,Y 91.188,Z 139.489,A -85,B 0,C 180,E1 -28791.132,E2 -28791.132} C_VEL
LIN {X 0,Y 91.573,Z 139.577,A -85,B 0,C 180,E1 -28798.232,E2 -28798.232} C_VEL
LIN {X 0,Y 92.698,Z 141.281,A -85,B 0,C 180,E1 -28803.939,E2 -28803.939} C_VEL
LIN {X 0,Y 94.891,Z 145.668,A -85,B 0,C 180,E1 -28810.484,E2 -28810.484} C_VEL
LIN {X 0,Y 96.968,Z 149.667,A -85,B 0,C 180,E1 -28814.795,E2 -28814.795} C_VEL
LIN {X 0,Y 100.065,Z 155.951,A -85,B 0,C 180,E1 -28819.855,E2 -28819.855} C_VEL
LIN {X 0,Y 101.449,Z 159.566,A -85,B 0,C 180,E1 -28821.891,E2 -28821.891} C_VEL
LIN {X 0,Y 102.866,Z 165.414,A -85,B 0,C 180,E1 -28824.088,E2 -28824.088} C_VEL
LIN {X 0,Y 102.587,Z 173.34,A -85,B 0,C 180,E1 -28824.894,E2 -28824.894} C_VEL
LIN {X 0,Y 99.715,Z 200.84,A -85,B 0,C 180,E1 -28826.188,E2 -28826.188} C_VEL
LIN {X 0,Y 97.03,Z 214.792,A -85,B 0,C 180,E1 -28827.375,E2 -28827.375} C_VEL
LIN {X 0,Y 93.327,Z 227.272,A -85,B 0,C 180,E1 -28828.902,E2 -28828.902} C_VEL
LIN {X 0,Y 88.47,Z 239.954,A -85,B 0,C 180,E1 -28831.35,E2 -28831.35} C_VEL
LIN {X 0,Y 82.974,Z 251.187,A -85,B 0,C 180,E1 -28834.324,E2 -28834.324} C_VEL
LIN {X 0,Y 77.895,Z 260.315,A -85,B 0,C 180,E1 -28837.862,E2 -28837.862} C_VEL
LIN {X 0,Y 71.744,Z 270.125,A -85,B 0,C 180,E1 -28843.291,E2 -28843.291} C_VEL
LIN {X 0,Y 67.709,Z 275.927,A -85,B 0,C 180,E1 -28847.568,E2 -28847.568} C_VEL
LIN {X 0,Y 62.51,Z 283.754,A -85,B 0,C 180,E1 -28855.792,E2 -28855.792} C_VEL
LIN {X 0,Y 58.562,Z 289.995,A -85,B 0,C 180,E1 -28865.16,E2 -28865.16} C_VEL
LIN {X 0,Y 56.346,Z 294.936,A -85,B 0,C 180,E1 -28875.552,E2 -28875.552} C_VEL
LIN {X 0,Y 55.929,Z 298.714,A -85,B 0,C 180,E1 -28886.395,E2 -28886.395} C_VEL
LIN {X 0,Y 56.141,Z 299.749,A -85,B 0,C 180,E1 -28889.997,E2 -28889.997} C_VEL
LIN {X 0,Y 55.983,Z 301.338,A -85,B 0,C 180,E1 -28897.209,E2 -28897.209} C_VEL
LIN {X 0,Y 57.803,Z 303.313,A -85,B 0,C 180,E1 -28911.39,E2 -28911.39} C_VEL
LIN {X 0,Y 59.916,Z 303.715,A -85,B 0,C 180,E1 -28917.979,E2 -28917.979} C_VEL
LIN {X 0,Y 66.416,Z 303.341,A -85,B 0,C 180,E1 -28929.41,E2 -28929.41} C_VEL
LIN {X 0,Y 75.088,Z 301.475,A -85,B 0,C 180,E1 -28938.482,E2 -28938.482} C_VEL
LIN {X 0,Y 80.006,Z 299.922,A -85,B 0,C 180,E1 -28942.238,E2 -28942.238} C_VEL
LIN {X 0,Y 87.97,Z 296.839,A -85,B 0,C 180,E1 -28947.016,E2 -28947.016} C_VEL
LIN {X 0,Y 96.525,Z 292.741,A -85,B 0,C 180,E1 -28950.891,E2 -28950.891} C_VEL
LIN {X 0,Y 107.06,Z 286.502,A -85,B 0,C 180,E1 -28954.501,E2 -28954.501} C_VEL
LIN {X 0,Y 116.35,Z 279.754,A -85,B 0,C 180,E1 -28957.093,E2 -28957.093} C_VEL
LIN {X 0,Y 124.319,Z 272.908,A -85,B 0,C 180,E1 -28958.868,E2 -28958.868} C_VEL
LIN {X 0,Y 130.769,Z 266.473,A -85,B 0,C 180,E1 -28960.135,E2 -28960.135} C_VEL
LIN {X 0,Y 138.95,Z 256.833,A -85,B 0,C 180,E1 -28961.504,E2 -28961.504} C_VEL
LIN {X 0,Y 146.423,Z 246.143,A -85,B 0,C 180,E1 -28962.542,E2 -28962.542} C_VEL
LIN {X 0,Y 152.278,Z 235.808,A -85,B 0,C 180,E1 -28963.265,E2 -28963.265} C_VEL
LIN {X 0,Y 157.384,Z 224.329,A -85,B 0,C 180,E1 -28963.895,E2 -28963.895} C_VEL
LIN {X 0,Y 160.198,Z 216.313,A -85,B 0,C 180,E1 -28964.234,E2 -28964.234} C_VEL
LIN {X 0,Y 160.491,Z 215.161,A -85,B 0,C 180,E1 -28964.445,E2 -28964.445} C_VEL
LIN {X 0,Y 160.421,Z 211.156,A -85,B 0,C 180,E1 -28967.669,E2 -28967.669} C_VEL
LIN {X 0,Y 160.258,Z 208.957,A -85,B 0,C 180,E1 -28971.171,E2 -28971.171} C_VEL
LIN {X 0,Y 160.211,Z 208.972,A -85,B 0,C 180,E1 -28976.324,E2 -28976.324} C_VEL
LIN {X 0,Y 160.348,Z 211.251,A -85,B 0,C 180,E1 -28980.001,E2 -28980.001} C_VEL
LIN {X 0,Y 160.5,Z 213.786,A -85,B 0,C 180,E1 -28982.667,E2 -28982.667} C_VEL
LIN {X 0,Y 156.164,Z 225.547,A -85,B 0,C 180,E1 -28983.37,E2 -28983.37} C_VEL
LIN {X 0,Y 150.648,Z 237.018,A -85,B 0,C 180,E1 -28984.318,E2 -28984.318} C_VEL
LIN {X 0,Y 147.491,Z 242.457,A -85,B 0,C 180,E1 -28984.849,E2 -28984.849} C_VEL
LIN {X 0,Y 144.257,Z 247.345,A -85,B 0,C 180,E1 -28985.153,E2 -28985.153} C_VEL
LIN {X 0,Y 138.06,Z 255.09,A -85,B 0,C 180,E1 -28985.011,E2 -28985.011} C_VEL
LIN {X 0,Y 131.308,Z 262.366,A -85,B 0,C 180,E1 -28984.933,E2 -28984.933} C_VEL
LIN {X 0,Y 127.205,Z 266.437,A -85,B 0,C 180,E1 -28985.405,E2 -28985.405} C_VEL
LIN {X 0,Y 118.655,Z 274.075,A -85,B 0,C 180,E1 -28987.214,E2 -28987.214} C_VEL
LIN {X 0,Y 108.726,Z 281.388,A -85,B 0,C 180,E1 -28989.693,E2 -28989.693} C_VEL
LIN {X 0,Y 100.632,Z 286.273,A -85,B 0,C 180,E1 -28992.118,E2 -28992.118} C_VEL
LIN {X 0,Y 91.229,Z 290.954,A -85,B 0,C 180,E1 -28995.65,E2 -28995.65} C_VEL
LIN {X 0,Y 81.812,Z 294.587,A -85,B 0,C 180,E1 -29000.099,E2 -29000.099} C_VEL
LIN {X 0,Y 76.476,Z 296.173,A -85,B 0,C 180,E1 -29003.228,E2 -29003.228} C_VEL
LIN {X 0,Y 71.061,Z 297.451,A -85,B 0,C 180,E1 -29007.119,E2 -29007.119} C_VEL
LIN {X 0,Y 64.673,Z 298.466,A -85,B 0,C 180,E1 -29012.914,E2 -29012.914} C_VEL
LIN {X 0,Y 57.324,Z 298.721,A -85,B 0,C 180,E1 -29022.645,E2 -29022.645} C_VEL
LIN {X 0,Y 52.164,Z 297.821,A -85,B 0,C 180,E1 -29033.941,E2 -29033.941} C_VEL
LIN {X 0,Y 49.398,Z 296.216,A -85,B 0,C 180,E1 -29044.737,E2 -29044.737} C_VEL
LIN {X 0,Y 48.43,Z 293.519,A -85,B 0,C 180,E1 -29057.431,E2 -29057.431} C_VEL
LIN {X 0,Y 49.641,Z 289.785,A -85,B 0,C 180,E1 -29070.003,E2 -29070.003} C_VEL
LIN {X 0,Y 52.561,Z 284.949,A -85,B 0,C 180,E1 -29081.573,E2 -29081.573} C_VEL
LIN {X 0,Y 57.018,Z 278.867,A -85,B 0,C 180,E1 -29091.704,E2 -29091.704} C_VEL
LIN {X 0,Y 62.829,Z 271.309,A -85,B 0,C 180,E1 -29100.226,E2 -29100.226} C_VEL
LIN {X 0,Y 68.535,Z 263.583,A -85,B 0,C 180,E1 -29106.134,E2 -29106.134} C_VEL
LIN {X 0,Y 74.746,Z 254.191,A -85,B 0,C 180,E1 -29111.164,E2 -29111.164} C_VEL
LIN {X 0,Y 80.649,Z 243.76,A -85,B 0,C 180,E1 -29115.078,E2 -29115.078} C_VEL
LIN {X 0,Y 86.03,Z 232.225,A -85,B 0,C 180,E1 -29118.2,E2 -29118.2} C_VEL
LIN {X 0,Y 90.718,Z 219.95,A -85,B 0,C 180,E1 -29120.344,E2 -29120.344} C_VEL
LIN {X 0,Y 94.426,Z 206.504,A -85,B 0,C 180,E1 -29122.004,E2 -29122.004} C_VEL
LIN {X 0,Y 96.758,Z 193.606,A -85,B 0,C 180,E1 -29123.035,E2 -29123.035} C_VEL
LIN {X 0,Y 99.567,Z 167.205,A -85,B 0,C 180,E1 -29124.183,E2 -29124.183} C_VEL
LIN {X 0,Y 98.987,Z 165.234,A -85,B 0,C 180,E1 -29125.126,E2 -29125.126} C_VEL
LIN {X 0,Y 96.673,Z 159.67,A -85,B 0,C 180,E1 -29128.93,E2 -29128.93} C_VEL
LIN {X 0,Y 94.496,Z 154.759,A -85,B 0,C 180,E1 -29133.284,E2 -29133.284} C_VEL
LIN {X 0,Y 92.728,Z 151.376,A -85,B 0,C 180,E1 -29137.73,E2 -29137.73} C_VEL
LIN {X 0,Y 91.255,Z 148.062,A -85,B 0,C 180,E1 -29143.337,E2 -29143.337} C_VEL
LIN {X 0,Y 90.312,Z 146.552,A -85,B 0,C 180,E1 -29151.045,E2 -29151.045} C_VEL
LIN {X 0,Y 90.638,Z 146.618,A -85,B 0,C 180,E1 -29157.883,E2 -29157.883} C_VEL
LIN {X 0,Y 91.468,Z 148.052,A -85,B 0,C 180,E1 -29162.702,E2 -29162.702} C_VEL
LIN {X 0,Y 93.351,Z 152.285,A -85,B 0,C 180,E1 -29169.142,E2 -29169.142} C_VEL
LIN {X 0,Y 95.503,Z 156.869,A -85,B 0,C 180,E1 -29174.05,E2 -29174.05} C_VEL
LIN {X 0,Y 97.806,Z 162.264,A -85,B 0,C 180,E1 -29178.22,E2 -29178.22} C_VEL
LIN {X 0,Y 98.639,Z 165.081,A -85,B 0,C 180,E1 -29179.679,E2 -29179.679} C_VEL
LIN {X 0,Y 99.286,Z 168.156,A -85,B 0,C 180,E1 -29180.889,E2 -29180.889} C_VEL
LIN {X 0,Y 99.016,Z 173.504,A -85,B 0,C 180,E1 -29181.412,E2 -29181.412} C_VEL
LIN {X 0,Y 96.011,Z 200.879,A -85,B 0,C 180,E1 -29182.658,E2 -29182.658} C_VEL
LIN {X 0,Y 93.183,Z 214.745,A -85,B 0,C 180,E1 -29183.784,E2 -29183.784} C_VEL
LIN {X 0,Y 89.342,Z 227.074,A -85,B 0,C 180,E1 -29185.222,E2 -29185.222} C_VEL
LIN {X 0,Y 84.245,Z 239.72,A -85,B 0,C 180,E1 -29187.575,E2 -29187.575} C_VEL
LIN {X 0,Y 78.461,Z 250.921,A -85,B 0,C 180,E1 -29190.439,E2 -29190.439} C_VEL
LIN {X 0,Y 73.063,Z 260.03,A -85,B 0,C 180,E1 -29193.934,E2 -29193.934} C_VEL
LIN {X 0,Y 66.411,Z 269.852,A -85,B 0,C 180,E1 -29199.415,E2 -29199.415} C_VEL
LIN {X 0,Y 61.548,Z 276.33,A -85,B 0,C 180,E1 -29204.462,E2 -29204.462} C_VEL
LIN {X 0,Y 55.88,Z 283.993,A -85,B 0,C 180,E1 -29213.313,E2 -29213.313} C_VEL
LIN {X 0,Y 51.027,Z 291.028,A -85,B 0,C 180,E1 -29225.591,E2 -29225.591} C_VEL
LIN {X 0,Y 49.031,Z 295.661,A -85,B 0,C 180,E1 -29237.581,E2 -29237.581} C_VEL
LIN {X 0,Y 49.041,Z 299.153,A -85,B 0,C 180,E1 -29249.997,E2 -29249.997} C_VEL
LIN {X 0,Y 48.957,Z 300.789,A -85,B 0,C 180,E1 -29258.25,E2 -29258.25} C_VEL
LIN {X 0,Y 51.239,Z 302.835,A -85,B 0,C 180,E1 -29274.295,E2 -29274.295} C_VEL
LIN {X 0,Y 53.715,Z 303.29,A -85,B 0,C 180,E1 -29281.554,E2 -29281.554} C_VEL
LIN {X 0,Y 61.076,Z 303.011,A -85,B 0,C 180,E1 -29293.66,E2 -29293.66} C_VEL
LIN {X 0,Y 70.557,Z 301.225,A -85,B 0,C 180,E1 -29302.828,E2 -29302.828} C_VEL
LIN {X 0,Y 75.846,Z 299.748,A -85,B 0,C 180,E1 -29306.503,E2 -29306.503} C_VEL
LIN {X 0,Y 84.312,Z 296.734,A -85,B 0,C 180,E1 -29311.071,E2 -29311.071} C_VEL
LIN {X 0,Y 93.277,Z 292.714,A -85,B 0,C 180,E1 -29314.704,E2 -29314.704} C_VEL
LIN {X 0,Y 104.205,Z 286.599,A -85,B 0,C 180,E1 -29318.022,E2 -29318.022} C_VEL
LIN {X 0,Y 113.778,Z 279.959,A -85,B 0,C 180,E1 -29320.383,E2 -29320.383} C_VEL
LIN {X 0,Y 121.943,Z 273.234,A -85,B 0,C 180,E1 -29321.977,E2 -29321.977} C_VEL
LIN {X 0,Y 128.535,Z 266.934,A -85,B 0,C 180,E1 -29323.105,E2 -29323.105} C_VEL
LIN {X 0,Y 136.873,Z 257.47,A -85,B 0,C 180,E1 -29324.309,E2 -29324.309} C_VEL
LIN {X 0,Y 144.463,Z 246.99,A -85,B 0,C 180,E1 -29325.213,E2 -29325.213} C_VEL
LIN {X 0,Y 151.248,Z 235.352,A -85,B 0,C 180,E1 -29325.923,E2 -29325.923} C_VEL
LIN {X 0,Y 156.106,Z 224.685,A -85,B 0,C 180,E1 -29326.441,E2 -29326.441} C_VEL
LIN {X 0,Y 157.775,Z 220.269,A -85,B 0,C 180,E1 -29326.624,E2 -29326.624} C_VEL
LIN {X 0,Y 158.084,Z 218.924,A -85,B 0,C 180,E1 -29327.157,E2 -29327.157} C_VEL
LIN {X 0,Y 158.094,Z 216.757,A -85,B 0,C 180,E1 -29329.758,E2 -29329.758} C_VEL
LIN {X 0,Y 158.081,Z 215.62,A -85,B 0,C 180,E1 -29332.336,E2 -29332.336} C_VEL
LIN {X 0,Y 158.018,Z 215.627,A -85,B 0,C 180,E1 -29334.897,E2 -29334.897} C_VEL
LIN {X 0,Y 157.955,Z 216.647,A -85,B 0,C 180,E1 -29337.45,E2 -29337.45} C_VEL
LIN {X 0,Y 157.941,Z 218.551,A -85,B 0,C 180,E1 -29340.319,E2 -29340.319} C_VEL
LIN {X 0,Y 153.757,Z 228.789,A -85,B 0,C 180,E1 -29340.974,E2 -29340.974} C_VEL
LIN {X 0,Y 147.666,Z 240.366,A -85,B 0,C 180,E1 -29341.897,E2 -29341.897} C_VEL
LIN {X 0,Y 139.888,Z 252.028,A -85,B 0,C 180,E1 -29343.134,E2 -29343.134} C_VEL
LIN {X 0,Y 132.171,Z 261.303,A -85,B 0,C 180,E1 -29344.454,E2 -29344.454} C_VEL
LIN {X 0,Y 127.205,Z 266.437,A -85,B 0,C 180,E1 -29345.405,E2 -29345.405} C_VEL
LIN {X 0,Y 122.924,Z 270.36,A -85,B 0,C 180,E1 -29345.94,E2 -29345.94} C_VEL
LIN {X 0,Y 115.087,Z 276.468,A -85,B 0,C 180,E1 -29346.101,E2 -29346.101} C_VEL
LIN {X 0,Y 106.827,Z 281.902,A -85,B 0,C 180,E1 -29346.388,E2 -29346.388} C_VEL
LIN {X 0,Y 101.914,Z 284.764,A -85,B 0,C 180,E1 -29347.239,E2 -29347.239} C_VEL
LIN {X 0,Y 92.757,Z 289.542,A -85,B 0,C 180,E1 -29349.951,E2 -29349.951} C_VEL
LIN {X 0,Y 83.127,Z 293.512,A -85,B 0,C 180,E1 -29353.532,E2 -29353.532} C_VEL
LIN {X 0,Y 73.873,Z 296.383,A -85,B 0,C 180,E1 -29357.95,E2 -29357.95} C_VEL
LIN {X 0,Y 68.005,Z 297.704,A -85,B 0,C 180,E1 -29361.554,E2 -29361.554} C_VEL
LIN {X 0,Y 60.104,Z 298.874,A -85,B 0,C 180,E1 -29367.888,E2 -29367.888} C_VEL
LIN {X 0,Y 52.587,Z 299.143,A -85,B 0,C 180,E1 -29376.696,E2 -29376.696} C_VEL
LIN {X 0,Y 45.904,Z 298.177,A -85,B 0,C 180,E1 -29389.957,E2 -29389.957} C_VEL
LIN {X 0,Y 42.905,Z 296.8,A -85,B 0,C 180,E1 -29400.571,E2 -29400.571} C_VEL
LIN {X 0,Y 41.336,Z 294.19,A -85,B 0,C 180,E1 -29415.228,E2 -29415.228} C_VEL
LIN {X 0,Y 42.413,Z 290.542,A -85,B 0,C 180,E1 -29430.003,E2 -29430.003} C_VEL
LIN {X 0,Y 45.55,Z 285.799,A -85,B 0,C 180,E1 -29443.385,E2 -29443.385} C_VEL
LIN {X 0,Y 50.445,Z 279.821,A -85,B 0,C 180,E1 -29454.709,E2 -29454.709} C_VEL
LIN {X 0,Y 56.772,Z 272.382,A -85,B 0,C 180,E1 -29463.856,E2 -29463.856} C_VEL
LIN {X 0,Y 62.933,Z 264.79,A -85,B 0,C 180,E1 -29469.954,E2 -29469.954} C_VEL
LIN {X 0,Y 69.577,Z 255.609,A -85,B 0,C 180,E1 -29475,E2 -29475} C_VEL
LIN {X 0,Y 75.826,Z 245.439,A -85,B 0,C 180,E1 -29478.86,E2 -29478.86} C_VEL
LIN {X 0,Y 81.476,Z 234.202,A -85,B 0,C 180,E1 -29481.919,E2 -29481.919} C_VEL
LIN {X 0,Y 86.312,Z 222.513,A -85,B 0,C 180,E1 -29484.017,E2 -29484.017} C_VEL
LIN {X 0,Y 90.348,Z 209.577,A -85,B 0,C 180,E1 -29485.565,E2 -29485.565} C_VEL
LIN {X 0,Y 93.065,Z 196.33,A -85,B 0,C 180,E1 -29486.674,E2 -29486.674} C_VEL
LIN {X 0,Y 96.057,Z 169.688,A -85,B 0,C 180,E1 -29487.923,E2 -29487.923} C_VEL
LIN {X 0,Y 93.996,Z 164.304,A -85,B 0,C 180,E1 -29491.988,E2 -29491.988} C_VEL
LIN {X 0,Y 92.339,Z 160.278,A -85,B 0,C 180,E1 -29496.028,E2 -29496.028} C_VEL
LIN {X 0,Y 91.213,Z 157.786,A -85,B 0,C 180,E1 -29499.48,E2 -29499.48} C_VEL
LIN {X 0,Y 90.136,Z 154.894,A -85,B 0,C 180,E1 -29504.414,E2 -29504.414} C_VEL
LIN {X 0,Y 89.433,Z 153.635,A -85,B 0,C 180,E1 -29510.956,E2 -29510.956} C_VEL
LIN {X 0,Y 89.682,Z 153.605,A -85,B 0,C 180,E1 -29517.272,E2 -29517.272} C_VEL
LIN {X 0,Y 90.321,Z 154.97,A -85,B 0,C 180,E1 -29521.671,E2 -29521.671} C_VEL
LIN {X 0,Y 91.81,Z 158.788,A -85,B 0,C 180,E1 -29527.594,E2 -29527.594} C_VEL
LIN {X 0,Y 93.523,Z 162.907,A -85,B 0,C 180,E1 -29532.122,E2 -29532.122} C_VEL
LIN {X 0,Y 95.429,Z 167.985,A -85,B 0,C 180,E1 -29536.137,E2 -29536.137} C_VEL
LIN {X 0,Y 95.992,Z 170.799,A -85,B 0,C 180,E1 -29537.411,E2 -29537.411} C_VEL
LIN {X 0,Y 95.506,Z 176.481,A -85,B 0,C 180,E1 -29537.793,E2 -29537.793} C_VEL
LIN {X 0,Y 92.702,Z 200.623,A -85,B 0,C 180,E1 -29538.836,E2 -29538.836} C_VEL
LIN {X 0,Y 89.824,Z 214.174,A -85,B 0,C 180,E1 -29539.854,E2 -29539.854} C_VEL
LIN {X 0,Y 85.758,Z 226.795,A -85,B 0,C 180,E1 -29541.216,E2 -29541.216} C_VEL
LIN {X 0,Y 80.423,Z 239.425,A -85,B 0,C 180,E1 -29543.421,E2 -29543.421} C_VEL
LIN {X 0,Y 74.352,Z 250.608,A -85,B 0,C 180,E1 -29546.103,E2 -29546.103} C_VEL
LIN {X 0,Y 68.62,Z 259.709,A -85,B 0,C 180,E1 -29549.472,E2 -29549.472} C_VEL
LIN {X 0,Y 61.394,Z 269.598,A -85,B 0,C 180,E1 -29554.914,E2 -29554.914} C_VEL
LIN {X 0,Y 55.599,Z 276.682,A -85,B 0,C 180,E1 -29560.67,E2 -29560.67} C_VEL
LIN {X 0,Y 49.367,Z 284.215,A -85,B 0,C 180,E1 -29570.158,E2 -29570.158} C_VEL
LIN {X 0,Y 44.62,Z 290.22,A -85,B 0,C 180,E1 -29581.798,E2 -29581.798} C_VEL
LIN {X 0,Y 42.096,Z 294.951,A -85,B 0,C 180,E1 -29595.493,E2 -29595.493} C_VEL
LIN {X 0,Y 41.925,Z 298.524,A -85,B 0,C 180,E1 -29609.997,E2 -29609.997} C_VEL
LIN {X 0,Y 41.936,Z 300.234,A -85,B 0,C 180,E1 -29619.644,E2 -29619.644} C_VEL
LIN {X 0,Y 44.852,Z 302.354,A -85,B 0,C 180,E1 -29638.036,E2 -29638.036} C_VEL
LIN {X 0,Y 51.628,Z 302.969,A -85,B 0,C 180,E1 -29652.89,E2 -29652.89} C_VEL
LIN {X 0,Y 61.122,Z 302.015,A -85,B 0,C 180,E1 -29663.594,E2 -29663.594} C_VEL
LIN {X 0,Y 72.159,Z 299.55,A -85,B 0,C 180,E1 -29671.226,E2 -29671.226} C_VEL
LIN {X 0,Y 81.108,Z 296.605,A -85,B 0,C 180,E1 -29675.477,E2 -29675.477} C_VEL
LIN {X 0,Y 90.474,Z 292.67,A -85,B 0,C 180,E1 -29678.768,E2 -29678.768} C_VEL
LIN {X 0,Y 100.135,Z 287.64,A -85,B 0,C 180,E1 -29681.346,E2 -29681.346} C_VEL
LIN {X 0,Y 109.932,Z 281.365,A -85,B 0,C 180,E1 -29683.523,E2 -29683.523} C_VEL
LIN {X 0,Y 118.255,Z 274.975,A -85,B 0,C 180,E1 -29684.955,E2 -29684.955} C_VEL
LIN {X 0,Y 126.659,Z 267.339,A -85,B 0,C 180,E1 -29686.171,E2 -29686.171} C_VEL
LIN {X 0,Y 135.134,Z 258.102,A -85,B 0,C 180,E1 -29687.193,E2 -29687.193} C_VEL
LIN {X 0,Y 142.825,Z 247.837,A -85,B 0,C 180,E1 -29687.951,E2 -29687.951} C_VEL
LIN {X 0,Y 149.69,Z 236.48,A -85,B 0,C 180,E1 -29688.542,E2 -29688.542} C_VEL
LIN {X 0,Y 154.996,Z 225.321,A -85,B 0,C 180,E1 -29689.01,E2 -29689.01} C_VEL
LIN {X 0,Y 155.527,Z 223.728,A -85,B 0,C 180,E1 -29689.587,E2 -29689.587} C_VEL
LIN {X 0,Y 155.602,Z 222.412,A -85,B 0,C 180,E1 -29692.213,E2 -29692.213} C_VEL
LIN {X 0,Y 155.543,Z 222.318,A -85,B 0,C 180,E1 -29694.816,E2 -29694.816} C_VEL
LIN {X 0,Y 155.363,Z 223.395,A -85,B 0,C 180,E1 -29697.408,E2 -29697.408} C_VEL
LIN {X 0,Y 154.695,Z 225.184,A -85,B 0,C 180,E1 -29698.134,E2 -29698.134} C_VEL
LIN {X 0,Y 148.97,Z 236.877,A -85,B 0,C 180,E1 -29698.871,E2 -29698.871} C_VEL
LIN {X 0,Y 142.138,Z 247.854,A -85,B 0,C 180,E1 -29699.802,E2 -29699.802} C_VEL
LIN {X 0,Y 135.266,Z 256.811,A -85,B 0,C 180,E1 -29700.752,E2 -29700.752} C_VEL
LIN {X 0,Y 126.587,Z 266.116,A -85,B 0,C 180,E1 -29702.117,E2 -29702.117} C_VEL
LIN {X 0,Y 118.454,Z 273.364,A -85,B 0,C 180,E1 -29703.566,E2 -29703.566} C_VEL
LIN {X 0,Y 107.731,Z 281.213,A -85,B 0,C 180,E1 -29705.828,E2 -29705.828} C_VEL
LIN {X 0,Y 101.914,Z 284.764,A -85,B 0,C 180,E1 -29707.239,E2 -29707.239} C_VEL
LIN {X 0,Y 96.888,Z 287.454,A -85,B 0,C 180,E1 -29708.225,E2 -29708.225} C_VEL
LIN {X 0,Y 84.192,Z 292.814,A -85,B 0,C 180,E1 -29709.344,E2 -29709.344} C_VEL
LIN {X 0,Y 76.857,Z 295.222,A -85,B 0,C 180,E1 -29710.53,E2 -29710.53} C_VEL
LIN {X 0,Y 73.386,Z 296.178,A -85,B 0,C 180,E1 -29711.712,E2 -29711.712} C_VEL
LIN {X 0,Y 65.649,Z 297.957,A -85,B 0,C 180,E1 -29715.538,E2 -29715.538} C_VEL
LIN {X 0,Y 56.018,Z 299.287,A -85,B 0,C 180,E1 -29722.111,E2 -29722.111} C_VEL
LIN {X 0,Y 48.526,Z 299.565,A -85,B 0,C 180,E1 -29729.667,E2 -29729.667} C_VEL
LIN {X 0,Y 39.89,Z 298.525,A -85,B 0,C 180,E1 -29744.812,E2 -29744.812} C_VEL
LIN {X 0,Y 36.722,Z 297.371,A -85,B 0,C 180,E1 -29754.964,E2 -29754.964} C_VEL
LIN {X 0,Y 34.336,Z 294.838,A -85,B 0,C 180,E1 -29772.124,E2 -29772.124} C_VEL
LIN {X 0,Y 35.182,Z 291.276,A -85,B 0,C 180,E1 -29790.004,E2 -29790.004} C_VEL
LIN {X 0,Y 38.604,Z 286.638,A -85,B 0,C 180,E1 -29805.852,E2 -29805.852} C_VEL
LIN {X 0,Y 45.13,Z 279.643,A -85,B 0,C 180,E1 -29820.409,E2 -29820.409} C_VEL
LIN {X 0,Y 52.283,Z 272.085,A -85,B 0,C 180,E1 -29829.684,E2 -29829.684} C_VEL
LIN {X 0,Y 59.034,Z 264.358,A -85,B 0,C 180,E1 -29835.589,E2 -29835.589} C_VEL
LIN {X 0,Y 66.438,Z 254.58,A -85,B 0,C 180,E1 -29840.515,E2 -29840.515} C_VEL
LIN {X 0,Y 72.834,Z 244.545,A -85,B 0,C 180,E1 -29843.917,E2 -29843.917} C_VEL
LIN {X 0,Y 78.833,Z 233.017,A -85,B 0,C 180,E1 -29846.701,E2 -29846.701} C_VEL
LIN {X 0,Y 83.912,Z 220.829,A -85,B 0,C 180,E1 -29848.539,E2 -29848.539} C_VEL
LIN {X 0,Y 87.909,Z 207.697,A -85,B 0,C 180,E1 -29849.906,E2 -29849.906} C_VEL
LIN {X 0,Y 90.484,Z 194.9,A -85,B 0,C 180,E1 -29850.814,E2 -29850.814} C_VEL
LIN {X 0,Y 92.999,Z 173.083,A -85,B 0,C 180,E1 -29851.704,E2 -29851.704} C_VEL
LIN {X 0,Y 91.122,Z 167.593,A -85,B 0,C 180,E1 -29856.603,E2 -29856.603} C_VEL
LIN {X 0,Y 89.857,Z 164.309,A -85,B 0,C 180,E1 -29861.012,E2 -29861.012} C_VEL
LIN {X 0,Y 88.997,Z 161.765,A -85,B 0,C 180,E1 -29865.775,E2 -29865.775} C_VEL
LIN {X 0,Y 88.555,Z 160.717,A -85,B 0,C 180,E1 -29870.866,E2 -29870.866} C_VEL
LIN {X 0,Y 88.754,Z 160.655,A -85,B 0,C 180,E1 -29876.886,E2 -29876.886} C_VEL
LIN {X 0,Y 89.201,Z 161.831,A -85,B 0,C 180,E1 -29880.563,E2 -29880.563} C_VEL
LIN {X 0,Y 90.345,Z 165.257,A -85,B 0,C 180,E1 -29885.999,E2 -29885.999} C_VEL
LIN {X 0,Y 91.724,Z 169.18,A -85,B 0,C 180,E1 -29890.317,E2 -29890.317} C_VEL
LIN {X 0,Y 93.044,Z 173.358,A -85,B 0,C 180,E1 -29893.652,E2 -29893.652} C_VEL
LIN {X 0,Y 89.921,Z 199.881,A -85,B 0,C 180,E1 -29894.736,E2 -29894.736} C_VEL
LIN {X 0,Y 86.904,Z 213.659,A -85,B 0,C 180,E1 -29895.657,E2 -29895.657} C_VEL
LIN {X 0,Y 83.049,Z 225.488,A -85,B 0,C 180,E1 -29896.795,E2 -29896.795} C_VEL
LIN {X 0,Y 77.836,Z 237.493,A -85,B 0,C 180,E1 -29898.54,E2 -29898.54} C_VEL
LIN {X 0,Y 71.514,Z 248.992,A -85,B 0,C 180,E1 -29900.991,E2 -29900.991} C_VEL
LIN {X 0,Y 64.65,Z 259.371,A -85,B 0,C 180,E1 -29904.429,E2 -29904.429} C_VEL
LIN {X 0,Y 56.683,Z 269.502,A -85,B 0,C 180,E1 -29909.777,E2 -29909.777} C_VEL
LIN {X 0,Y 51.2,Z 275.634,A -85,B 0,C 180,E1 -29914.549,E2 -29914.549} C_VEL
LIN {X 0,Y 44.104,Z 283.287,A -85,B 0,C 180,E1 -29924.182,E2 -29924.182} C_VEL
LIN {X 0,Y 38.481,Z 289.398,A -85,B 0,C 180,E1 -29936.772,E2 -29936.772} C_VEL
LIN {X 0,Y 35.223,Z 294.221,A -85,B 0,C 180,E1 -29952.58,E2 -29952.58} C_VEL
LIN {X 0,Y 34.814,Z 297.883,A -85,B 0,C 180,E1 -29969.996,E2 -29969.996} C_VEL
LIN {X 0,Y 34.951,Z 299.657,A -85,B 0,C 180,E1 -29981.596,E2 -29981.596} C_VEL
LIN {X 0,Y 38.707,Z 301.871,A -85,B 0,C 180,E1 -30003,E2 -30003} C_VEL
LIN {X 0,Y 46.672,Z 302.57,A -85,B 0,C 180,E1 -30018.839,E2 -30018.839} C_VEL
LIN {X 0,Y 51.696,Z 302.351,A -85,B 0,C 180,E1 -30024.651,E2 -30024.651} C_VEL
LIN {X 0,Y 62.969,Z 300.721,A -85,B 0,C 180,E1 -30033.233,E2 -30033.233} C_VEL
LIN {X 0,Y 75.245,Z 297.558,A -85,B 0,C 180,E1 -30039.064,E2 -30039.064} C_VEL
LIN {X 0,Y 84.876,Z 294.046,A -85,B 0,C 180,E1 -30042.213,E2 -30042.213} C_VEL
LIN {X 0,Y 94.76,Z 289.486,A -85,B 0,C 180,E1 -30044.608,E2 -30044.608} C_VEL
LIN {X 0,Y 106.456,Z 282.635,A -85,B 0,C 180,E1 -30046.839,E2 -30046.839} C_VEL
LIN {X 0,Y 114.898,Z 276.599,A -85,B 0,C 180,E1 -30048.141,E2 -30048.141} C_VEL
LIN {X 0,Y 125.156,Z 267.732,A -85,B 0,C 180,E1 -30049.318,E2 -30049.318} C_VEL
LIN {X 0,Y 133.746,Z 258.667,A -85,B 0,C 180,E1 -30050.144,E2 -30050.144} C_VEL
LIN {X 0,Y 141.521,Z 248.681,A -85,B 0,C 180,E1 -30050.746,E2 -30050.746} C_VEL
LIN {X 0,Y 148.479,Z 237.55,A -85,B 0,C 180,E1 -30051.212,E2 -30051.212} C_VEL
LIN {X 0,Y 152.012,Z 230.747,A -85,B 0,C 180,E1 -30051.449,E2 -30051.449} C_VEL
LIN {X 0,Y 152.744,Z 229.085,A -85,B 0,C 180,E1 -30052.066,E2 -30052.066} C_VEL
LIN {X 0,Y 152.702,Z 228.865,A -85,B 0,C 180,E1 -30054.719,E2 -30054.719} C_VEL
LIN {X 0,Y 152.564,Z 229.217,A -85,B 0,C 180,E1 -30055.625,E2 -30055.625} C_VEL
LIN {X 0,Y 146.117,Z 241.12,A -85,B 0,C 180,E1 -30056.394,E2 -30056.394} C_VEL
LIN {X 0,Y 138.714,Z 251.946,A -85,B 0,C 180,E1 -30057.255,E2 -30057.255} C_VEL
LIN {X 0,Y 130.072,Z 262.065,A -85,B 0,C 180,E1 -30058.298,E2 -30058.298} C_VEL
LIN {X 0,Y 121.234,Z 270.507,A -85,B 0,C 180,E1 -30059.532,E2 -30059.532} C_VEL
LIN {X 0,Y 110.715,Z 278.711,A -85,B 0,C 180,E1 -30061.261,E2 -30061.261} C_VEL
LIN {X 0,Y 102.039,Z 284.213,A -85,B 0,C 180,E1 -30062.952,E2 -30062.952} C_VEL
LIN {X 0,Y 91.769,Z 289.54,A -85,B 0,C 180,E1 -30065.404,E2 -30065.404} C_VEL
LIN {X 0,Y 81.713,Z 293.619,A -85,B 0,C 180,E1 -30068.481,E2 -30068.481} C_VEL
LIN {X 0,Y 73.386,Z 296.178,A -85,B 0,C 180,E1 -30071.712,E2 -30071.712} C_VEL
LIN {X 0,Y 68.091,Z 297.475,A -85,B 0,C 180,E1 -30073.578,E2 -30073.578} C_VEL
LIN {X 0,Y 58.621,Z 299.114,A -85,B 0,C 180,E1 -30075.859,E2 -30075.859} C_VEL
LIN {X 0,Y 49.182,Z 299.921,A -85,B 0,C 180,E1 -30079.019,E2 -30079.019} C_VEL
LIN {X 0,Y 44.118,Z 299.913,A -85,B 0,C 180,E1 -30082.773,E2 -30082.773} C_VEL
LIN {X 0,Y 34.957,Z 299.006,A -85,B 0,C 180,E1 -30096.476,E2 -30096.476} C_VEL
LIN {X 0,Y 30.995,Z 297.917,A -85,B 0,C 180,E1 -30107.145,E2 -30107.145} C_VEL
LIN {X 0,Y 28.243,Z 296.405,A -85,B 0,C 180,E1 -30120.159,E2 -30120.159} C_VEL
LIN {X 0,Y 27.31,Z 293.282,A -85,B 0,C 180,E1 -30142.613,E2 -30142.613} C_VEL
LIN {X 0,Y 30.155,Z 289.094,A -85,B 0,C 180,E1 -30163.482,E2 -30163.482} C_VEL
LIN {X 0,Y 36.796,Z 282.728,A -85,B 0,C 180,E1 -30181.69,E2 -30181.69} C_VEL
LIN {X 0,Y 44.279,Z 275.83,A -85,B 0,C 180,E1 -30192.425,E2 -30192.425} C_VEL
LIN {X 0,Y 51.333,Z 268.786,A -85,B 0,C 180,E1 -30198.856,E2 -30198.856} C_VEL
LIN {X 0,Y 58.797,Z 260.309,A -85,B 0,C 180,E1 -30203.791,E2 -30203.791} C_VEL
LIN {X 0,Y 66.517,Z 249.848,A -85,B 0,C 180,E1 -30207.704,E2 -30207.704} C_VEL
LIN {X 0,Y 72.801,Z 239.516,A -85,B 0,C 180,E1 -30210.328,E2 -30210.328} C_VEL
LIN {X 0,Y 78.388,Z 228.21,A -85,B 0,C 180,E1 -30212.3,E2 -30212.3} C_VEL
LIN {X 0,Y 83.167,Z 215.776,A -85,B 0,C 180,E1 -30213.623,E2 -30213.623} C_VEL
LIN {X 0,Y 86.705,Z 202.546,A -85,B 0,C 180,E1 -30214.686,E2 -30214.686} C_VEL
LIN {X 0,Y 88.85,Z 189.592,A -85,B 0,C 180,E1 -30215.323,E2 -30215.323} C_VEL
LIN {X 0,Y 90.301,Z 176.614,A -85,B 0,C 180,E1 -30215.836,E2 -30215.836} C_VEL
LIN {X 0,Y 89.157,Z 172.681,A -85,B 0,C 180,E1 -30219.896,E2 -30219.896} C_VEL
LIN {X 0,Y 88.411,Z 170.468,A -85,B 0,C 180,E1 -30223.378,E2 -30223.378} C_VEL
LIN {X 0,Y 87.912,Z 168.519,A -85,B 0,C 180,E1 -30227.26,E2 -30227.26} C_VEL
LIN {X 0,Y 87.648,Z 167.666,A -85,B 0,C 180,E1 -30232.637,E2 -30232.637} C_VEL
LIN {X 0,Y 87.862,Z 167.753,A -85,B 0,C 180,E1 -30236.855,E2 -30236.855} C_VEL
LIN {X 0,Y 88.132,Z 168.762,A -85,B 0,C 180,E1 -30239.575,E2 -30239.575} C_VEL
LIN {X 0,Y 89.019,Z 171.993,A -85,B 0,C 180,E1 -30244.669,E2 -30244.669} C_VEL
LIN {X 0,Y 90.22,Z 176.205,A -85,B 0,C 180,E1 -30249.103,E2 -30249.103} C_VEL
LIN {X 0,Y 90.378,Z 176.944,A -85,B 0,C 180,E1 -30249.645,E2 -30249.645} C_VEL
LIN {X 0,Y 87.63,Z 199.155,A -85,B 0,C 180,E1 -30250.41,E2 -30250.41} C_VEL
LIN {X 0,Y 84.647,Z 212.526,A -85,B 0,C 180,E1 -30251.15,E2 -30251.15} C_VEL
LIN {X 0,Y 80.809,Z 224.179,A -85,B 0,C 180,E1 -30252.067,E2 -30252.067} C_VEL
LIN {X 0,Y 75.854,Z 235.555,A -85,B 0,C 180,E1 -30253.376,E2 -30253.376} C_VEL
LIN {X 0,Y 70.902,Z 244.682,A -85,B 0,C 180,E1 -30254.877,E2 -30254.877} C_VEL
LIN {X 0,Y 64.436,Z 254.715,A -85,B 0,C 180,E1 -30257.371,E2 -30257.371} C_VEL
LIN {X 0,Y 56.543,Z 264.814,A -85,B 0,C 180,E1 -30261.211,E2 -30261.211} C_VEL
LIN {X 0,Y 50.464,Z 271.506,A -85,B 0,C 180,E1 -30264.987,E2 -30264.987} C_VEL
LIN {X 0,Y 41.972,Z 279.931,A -85,B 0,C 180,E1 -30273.146,E2 -30273.146} C_VEL
LIN {X 0,Y 34.747,Z 286.662,A -85,B 0,C 180,E1 -30284.928,E2 -30284.928} C_VEL
LIN {X 0,Y 29.553,Z 292.003,A -85,B 0,C 180,E1 -30301.594,E2 -30301.594} C_VEL
LIN {X 0,Y 27.576,Z 296.135,A -85,B 0,C 180,E1 -30322.674,E2 -30322.674} C_VEL
LIN {X 0,Y 27.701,Z 297.243,A -85,B 0,C 180,E1 -30329.995,E2 -30329.995} C_VEL
LIN {X 0,Y 28.027,Z 299.059,A -85,B 0,C 180,E1 -30344.517,E2 -30344.517} C_VEL
LIN {X 0,Y 29.758,Z 300.438,A -85,B 0,C 180,E1 -30358.181,E2 -30358.181} C_VEL
LIN {X 0,Y 37.208,Z 301.957,A -85,B 0,C 180,E1 -30379.066,E2 -30379.066} C_VEL
LIN {X 0,Y 47.923,Z 301.999,A -85,B 0,C 180,E1 -30391.625,E2 -30391.625} C_VEL
LIN {X 0,Y 53.907,Z 301.436,A -85,B 0,C 180,E1 -30395.862,E2 -30395.862} C_VEL
LIN {X 0,Y 66.479,Z 299.126,A -85,B 0,C 180,E1 -30402.066,E2 -30402.066} C_VEL
LIN {X 0,Y 76.309,Z 296.345,A -85,B 0,C 180,E1 -30405.242,E2 -30405.242} C_VEL
LIN {X 0,Y 86.348,Z 292.582,A -85,B 0,C 180,E1 -30407.6,E2 -30407.6} C_VEL
LIN {X 0,Y 96.535,Z 287.736,A -85,B 0,C 180,E1 -30409.359,E2 -30409.359} C_VEL
LIN {X 0,Y 108.506,Z 280.541,A -85,B 0,C 180,E1 -30411.013,E2 -30411.013} C_VEL
LIN {X 0,Y 117.122,Z 274.142,A -85,B 0,C 180,E1 -30411.918,E2 -30411.918} C_VEL
LIN {X 0,Y 125.778,Z 266.494,A -85,B 0,C 180,E1 -30412.648,E2 -30412.648} C_VEL
LIN {X 0,Y 134.464,Z 257.236,A -85,B 0,C 180,E1 -30413.239,E2 -30413.239} C_VEL
LIN {X 0,Y 141.427,Z 248.243,A -85,B 0,C 180,E1 -30413.64,E2 -30413.64} C_VEL
LIN {X 0,Y 141.318,Z 248.36,A -85,B 0,C 180,E1 -30414.052,E2 -30414.052} C_VEL
LIN {X 0,Y 133.198,Z 258.537,A -85,B 0,C 180,E1 -30414.805,E2 -30414.805} C_VEL
LIN {X 0,Y 125.101,Z 266.88,A -85,B 0,C 180,E1 -30415.673,E2 -30415.673} C_VEL
LIN {X 0,Y 115.009,Z 275.412,A -85,B 0,C 180,E1 -30416.895,E2 -30416.895} C_VEL
LIN {X 0,Y 105.466,Z 281.98,A -85,B 0,C 180,E1 -30418.251,E2 -30418.251} C_VEL
LIN {X 0,Y 95.167,Z 287.731,A -85,B 0,C 180,E1 -30420.001,E2 -30420.001} C_VEL
LIN {X 0,Y 84.408,Z 292.445,A -85,B 0,C 180,E1 -30422.409,E2 -30422.409} C_VEL
LIN {X 0,Y 73.676,Z 295.97,A -85,B 0,C 180,E1 -30425.475,E2 -30425.475} C_VEL
LIN {X 0,Y 64.064,Z 298.21,A -85,B 0,C 180,E1 -30429.145,E2 -30429.145} C_VEL
LIN {X 0,Y 52.625,Z 299.697,A -85,B 0,C 180,E1 -30435.494,E2 -30435.494} C_VEL
LIN {X 0,Y 44.118,Z 299.913,A -85,B 0,C 180,E1 -30442.773,E2 -30442.773} C_VEL
LIN {X 0,Y 39.281,Z 299.723,A -85,B 0,C 180,E1 -30447.423,E2 -30447.423} C_VEL
LIN {X 0,Y 30.739,Z 298.864,A -85,B 0,C 180,E1 -30455.616,E2 -30455.616} C_VEL
LIN {X 0,Y 24.492,Z 297.599,A -85,B 0,C 180,E1 -30465.654,E2 -30465.654} C_VEL
LIN {X 0,Y 21.226,Z 296.3,A -85,B 0,C 180,E1 -30477.712,E2 -30477.712} C_VEL
LIN {X 0,Y 20.632,Z 295.754,A -85,B 0,C 180,E1 -30482.709,E2 -30482.709} C_VEL
LIN {X 0,Y 21.175,Z 291.991,A -85,B 0,C 180,E1 -30515.25,E2 -30515.25} C_VEL
LIN {X 0,Y 25.064,Z 288.245,A -85,B 0,C 180,E1 -30534.879,E2 -30534.879} C_VEL
LIN {X 0,Y 32.237,Z 282.606,A -85,B 0,C 180,E1 -30550.853,E2 -30550.853} C_VEL
LIN {X 0,Y 40.778,Z 275.592,A -85,B 0,C 180,E1 -30560.862,E2 -30560.862} C_VEL
LIN {X 0,Y 50.096,Z 266.781,A -85,B 0,C 180,E1 -30567.33,E2 -30567.33} C_VEL
LIN {X 0,Y 58.871,Z 256.899,A -85,B 0,C 180,E1 -30571.475,E2 -30571.475} C_VEL
LIN {X 0,Y 65.517,Z 247.859,A -85,B 0,C 180,E1 -30573.952,E2 -30573.952} C_VEL
LIN {X 0,Y 72.033,Z 236.969,A -85,B 0,C 180,E1 -30576.166,E2 -30576.166} C_VEL
LIN {X 0,Y 77.638,Z 225.254,A -85,B 0,C 180,E1 -30577.643,E2 -30577.643} C_VEL
LIN {X 0,Y 82.035,Z 213.302,A -85,B 0,C 180,E1 -30578.57,E2 -30578.57} C_VEL
LIN {X 0,Y 85.333,Z 200.302,A -85,B 0,C 180,E1 -30579.38,E2 -30579.38} C_VEL
LIN {X 0,Y 87.683,Z 184.077,A -85,B 0,C 180,E1 -30579.942,E2 -30579.942} C_VEL
LIN {X 0,Y 88.089,Z 180.391,A -85,B 0,C 180,E1 -30580.138,E2 -30580.138} C_VEL
LIN {X 0,Y 87.39,Z 177.603,A -85,B 0,C 180,E1 -30583.878,E2 -30583.878} C_VEL
LIN {X 0,Y 86.922,Z 175.421,A -85,B 0,C 180,E1 -30588.259,E2 -30588.259} C_VEL
LIN {X 0,Y 86.768,Z 174.722,A -85,B 0,C 180,E1 -30592.562,E2 -30592.562} C_VEL
LIN {X 0,Y 86.918,Z 174.691,A -85,B 0,C 180,E1 -30596.091,E2 -30596.091} C_VEL
LIN {X 0,Y 87.102,Z 175.792,A -85,B 0,C 180,E1 -30598.711,E2 -30598.711} C_VEL
LIN {X 0,Y 87.716,Z 178.622,A -85,B 0,C 180,E1 -30603.157,E2 -30603.157} C_VEL
LIN {X 0,Y 88.139,Z 180.486,A -85,B 0,C 180,E1 -30605.283,E2 -30605.283} C_VEL
LIN {X 0,Y 85.638,Z 199.626,A -85,B 0,C 180,E1 -30605.917,E2 -30605.917} C_VEL
LIN {X 0,Y 82.455,Z 213.137,A -85,B 0,C 180,E1 -30606.521,E2 -30606.521} C_VEL
LIN {X 0,Y 78.619,Z 224.279,A -85,B 0,C 180,E1 -30607.221,E2 -30607.221} C_VEL
LIN {X 0,Y 73.671,Z 235.241,A -85,B 0,C 180,E1 -30608.203,E2 -30608.203} C_VEL
LIN {X 0,Y 68.563,Z 244.359,A -85,B 0,C 180,E1 -30609.376,E2 -30609.376} C_VEL
LIN {X 0,Y 61.833,Z 254.376,A -85,B 0,C 180,E1 -30611.372,E2 -30611.372} C_VEL
LIN {X 0,Y 54.363,Z 263.564,A -85,B 0,C 180,E1 -30614.154,E2 -30614.154} C_VEL
LIN {X 0,Y 47.004,Z 271.225,A -85,B 0,C 180,E1 -30617.697,E2 -30617.697} C_VEL
LIN {X 0,Y 38.517,Z 278.945,A -85,B 0,C 180,E1 -30624.164,E2 -30624.164} C_VEL
LIN {X 0,Y 30.131,Z 285.79,A -85,B 0,C 180,E1 -30635.27,E2 -30635.27} C_VEL
LIN {X 0,Y 23.509,Z 291.226,A -85,B 0,C 180,E1 -30653.273,E2 -30653.273} C_VEL
LIN {X 0,Y 20.515,Z 295.449,A -85,B 0,C 180,E1 -30680.13,E2 -30680.13} C_VEL
LIN {X 0,Y 20.597,Z 296.603,A -85,B 0,C 180,E1 -30689.993,E2 -30689.993} C_VEL
LIN {X 0,Y 21.238,Z 298.462,A -85,B 0,C 180,E1 -30709.317,E2 -30709.317} C_VEL
LIN {X 0,Y 23.731,Z 299.889,A -85,B 0,C 180,E1 -30726.312,E2 -30726.312} C_VEL
LIN {X 0,Y 27.841,Z 300.904,A -85,B 0,C 180,E1 -30739.219,E2 -30739.219} C_VEL
LIN {X 0,Y 38.798,Z 301.758,A -85,B 0,C 180,E1 -30754.911,E2 -30754.911} C_VEL
LIN {X 0,Y 51.402,Z 301.134,A -85,B 0,C 180,E1 -30763.142,E2 -30763.142} C_VEL
LIN {X 0,Y 64.642,Z 298.914,A -85,B 0,C 180,E1 -30768.086,E2 -30768.086} C_VEL
LIN {X 0,Y 78.234,Z 295.122,A -85,B 0,C 180,E1 -30771.164,E2 -30771.164} C_VEL
LIN {X 0,Y 88.556,Z 291.093,A -85,B 0,C 180,E1 -30772.748,E2 -30772.748} C_VEL
LIN {X 0,Y 98.94,Z 285.958,A -85,B 0,C 180,E1 -30773.954,E2 -30773.954} C_VEL
LIN {X 0,Y 102.139,Z 284.073,A -85,B 0,C 180,E1 -30774.721,E2 -30774.721} C_VEL
LIN {X 0,Y 91.568,Z 289.494,A -85,B 0,C 180,E1 -30776.153,E2 -30776.153} C_VEL
LIN {X 0,Y 80.866,Z 293.769,A -85,B 0,C 180,E1 -30778.061,E2 -30778.061} C_VEL
LIN {X 0,Y 70.28,Z 296.911,A -85,B 0,C 180,E1 -30780.477,E2 -30780.477} C_VEL
LIN {X 0,Y 63.31,Z 298.444,A -85,B 0,C 180,E1 -30782.513,E2 -30782.513} C_VEL
LIN {X 0,Y 56.442,Z 299.498,A -85,B 0,C 180,E1 -30785.073,E2 -30785.073} C_VEL
LIN {X 0,Y 49.706,Z 300.127,A -85,B 0,C 180,E1 -30788.234,E2 -30788.234} C_VEL
LIN {X 0,Y 39.995,Z 300.256,A -85,B 0,C 180,E1 -30794.903,E2 -30794.903} C_VEL
LIN {X 0,Y 29.437,Z 299.226,A -85,B 0,C 180,E1 -30808.526,E2 -30808.526} C_VEL
LIN {X 0,Y 22.195,Z 297.014,A -85,B 0,C 180,E1 -30830.716,E2 -30830.716} C_VEL
LIN {X 0,Y 20.632,Z 295.754,A -85,B 0,C 180,E1 -30842.709,E2 -30842.709} C_VEL
LIN {X 0,Y 19.403,Z 294.135,A -85,B 0,C 180,E1 -30858.643,E2 -30858.643} C_VEL
LIN {X 0,Y 18.97,Z 290.93,A -85,B 0,C 180,E1 -30886.985,E2 -30886.985} C_VEL
LIN {X 0,Y 22.373,Z 286.998,A -85,B 0,C 180,E1 -30910.92,E2 -30910.92} C_VEL
LIN {X 0,Y 26.216,Z 284.19,A -85,B 0,C 180,E1 -30919.435,E2 -30919.435} C_VEL
LIN {X 0,Y 36.704,Z 276.607,A -85,B 0,C 180,E1 -30929.51,E2 -30929.51} C_VEL
LIN {X 0,Y 44.969,Z 269.562,A -85,B 0,C 180,E1 -30933.987,E2 -30933.987} C_VEL
LIN {X 0,Y 54.245,Z 260.088,A -85,B 0,C 180,E1 -30937.482,E2 -30937.482} C_VEL
LIN {X 0,Y 62.689,Z 249.45,A -85,B 0,C 180,E1 -30939.875,E2 -30939.875} C_VEL
LIN {X 0,Y 69.474,Z 238.881,A -85,B 0,C 180,E1 -30941.514,E2 -30941.514} C_VEL
LIN {X 0,Y 75.317,Z 227.424,A -85,B 0,C 180,E1 -30942.676,E2 -30942.676} C_VEL
LIN {X 0,Y 80.105,Z 215.14,A -85,B 0,C 180,E1 -30943.373,E2 -30943.373} C_VEL
LIN {X 0,Y 83.673,Z 202.122,A -85,B 0,C 180,E1 -30944.017,E2 -30944.017} C_VEL
LIN {X 0,Y 85.822,Z 189.055,A -85,B 0,C 180,E1 -30944.434,E2 -30944.434} C_VEL
LIN {X 0,Y 86.328,Z 184.625,A -85,B 0,C 180,E1 -30944.689,E2 -30944.689} C_VEL
LIN {X 0,Y 85.963,Z 182.326,A -85,B 0,C 180,E1 -30949.237,E2 -30949.237} C_VEL
LIN {X 0,Y 85.988,Z 181.65,A -85,B 0,C 180,E1 -30955.311,E2 -30955.311} C_VEL
LIN {X 0,Y 86.125,Z 183.059,A -85,B 0,C 180,E1 -30958.282,E2 -30958.282} C_VEL
LIN {X 0,Y 86.381,Z 184.65,A -85,B 0,C 180,E1 -30960.836,E2 -30960.836} C_VEL
LIN {X 0,Y 84.163,Z 200.249,A -85,B 0,C 180,E1 -30961.23,E2 -30961.23} C_VEL
LIN {X 0,Y 80.868,Z 213.615,A -85,B 0,C 180,E1 -30961.694,E2 -30961.694} C_VEL
LIN {X 0,Y 76.487,Z 225.597,A -85,B 0,C 180,E1 -30962.175,E2 -30962.175} C_VEL
LIN {X 0,Y 70.386,Z 238.156,A -85,B 0,C 180,E1 -30963.109,E2 -30963.109} C_VEL
LIN {X 0,Y 63.421,Z 249.288,A -85,B 0,C 180,E1 -30964.153,E2 -30964.153} C_VEL
LIN {X 0,Y 56.511,Z 258.355,A -85,B 0,C 180,E1 -30965.748,E2 -30965.748} C_VEL
LIN {X 0,Y 47.307,Z 268.251,A -85,B 0,C 180,E1 -30968.542,E2 -30968.542} C_VEL
LIN {X 0,Y 39.493,Z 275.262,A -85,B 0,C 180,E1 -30971.812,E2 -30971.812} C_VEL
LIN {X 0,Y 29.766,Z 282.775,A -85,B 0,C 180,E1 -30979.175,E2 -30979.175} C_VEL
LIN {X 0,Y 20.843,Z 288.762,A -85,B 0,C 180,E1 -30992.532,E2 -30992.532} C_VEL
LIN {X 0,Y 14.464,Z 293.474,A -85,B 0,C 180,E1 -31020.917,E2 -31020.917} C_VEL
LIN {X 0,Y 13.481,Z 295.962,A -85,B 0,C 180,E1 -31049.989,E2 -31049.989} C_VEL
LIN {X 0,Y 14.711,Z 297.862,A -85,B 0,C 180,E1 -31078.526,E2 -31078.526} C_VEL
LIN {X 0,Y 23.806,Z 300.408,A -85,B 0,C 180,E1 -31112.318,E2 -31112.318} C_VEL
LIN {X 0,Y 29.876,Z 301.069,A -85,B 0,C 180,E1 -31120.2,E2 -31120.2} C_VEL
LIN {X 0,Y 43.016,Z 301.264,A -85,B 0,C 180,E1 -31128.585,E2 -31128.585} C_VEL
LIN {X 0,Y 56.649,Z 299.964,A -85,B 0,C 180,E1 -31132.956,E2 -31132.956} C_VEL
LIN {X 0,Y 63.554,Z 298.702,A -85,B 0,C 180,E1 -31134.387,E2 -31134.387} C_VEL
LIN {X 0,Y 63.418,Z 298.654,A -85,B 0,C 180,E1 -31135.821,E2 -31135.821} C_VEL
LIN {X 0,Y 56.273,Z 299.792,A -85,B 0,C 180,E1 -31137.543,E2 -31137.543} C_VEL
LIN {X 0,Y 48.313,Z 300.517,A -85,B 0,C 180,E1 -31140.002,E2 -31140.002} C_VEL
LIN {X 0,Y 35.36,Z 300.596,A -85,B 0,C 180,E1 -31146.43,E2 -31146.43} C_VEL
LIN {X 0,Y 25.627,Z 299.576,A -85,B 0,C 180,E1 -31155.921,E2 -31155.921} C_VEL
LIN {X 0,Y 17.17,Z 297.599,A -85,B 0,C 180,E1 -31175.067,E2 -31175.067} C_VEL
LIN {X 0,Y 12.988,Z 294.642,A -85,B 0,C 180,E1 -31214.314,E2 -31214.314} C_VEL
LIN {X 0,Y 16.499,Z 290.631,A -85,B 0,C 180,E1 -31255.222,E2 -31255.222} C_VEL
LIN {X 0,Y 24.255,Z 285.509,A -85,B 0,C 180,E1 -31276.426,E2 -31276.426} C_VEL
LIN {X 0,Y 26.216,Z 284.19,A -85,B 0,C 180,E1 -31279.435,E2 -31279.435} C_VEL
LIN {X 0,Y 30.268,Z 281.228,A -85,B 0,C 180,E1 -31285.643,E2 -31285.643} C_VEL
LIN {X 0,Y 36.527,Z 275.99,A -85,B 0,C 180,E1 -31295.295,E2 -31295.295} C_VEL
LIN {X 0,Y 43.088,Z 270.116,A -85,B 0,C 180,E1 -31301.989,E2 -31301.989} C_VEL
LIN {X 0,Y 47.302,Z 266.15,A -85,B 0,C 180,E1 -31303.834,E2 -31303.834} C_VEL
LIN {X 0,Y 56.447,Z 256.316,A -85,B 0,C 180,E1 -31305.476,E2 -31305.476} C_VEL
LIN {X 0,Y 64.141,Z 246.06,A -85,B 0,C 180,E1 -31306.67,E2 -31306.67} C_VEL
LIN {X 0,Y 71.038,Z 234.601,A -85,B 0,C 180,E1 -31307.685,E2 -31307.685} C_VEL
LIN {X 0,Y 76.561,Z 222.811,A -85,B 0,C 180,E1 -31308.239,E2 -31308.239} C_VEL
LIN {X 0,Y 80.852,Z 210.401,A -85,B 0,C 180,E1 -31308.626,E2 -31308.626} C_VEL
LIN {X 0,Y 83.954,Z 197.108,A -85,B 0,C 180,E1 -31309.004,E2 -31309.004} C_VEL
LIN {X 0,Y 85.048,Z 189.638,A -85,B 0,C 180,E1 -31309.238,E2 -31309.238} C_VEL
LIN {X 0,Y 85.01,Z 188.809,A -85,B 0,C 180,E1 -31312.793,E2 -31312.793} C_VEL
LIN {X 0,Y 85.083,Z 189.014,A -85,B 0,C 180,E1 -31315.541,E2 -31315.541} C_VEL
LIN {X 0,Y 85.09,Z 189.4,A -85,B 0,C 180,E1 -31316.228,E2 -31316.228} C_VEL
LIN {X 0,Y 82.907,Z 202.687,A -85,B 0,C 180,E1 -31316.453,E2 -31316.453} C_VEL
LIN {X 0,Y 79.33,Z 215.637,A -85,B 0,C 180,E1 -31316.752,E2 -31316.752} C_VEL
LIN {X 0,Y 74.338,Z 228.322,A -85,B 0,C 180,E1 -31316.993,E2 -31316.993} C_VEL
LIN {X 0,Y 68.594,Z 239.424,A -85,B 0,C 180,E1 -31317.431,E2 -31317.431} C_VEL
LIN {X 0,Y 61.543,Z 250.138,A -85,B 0,C 180,E1 -31317.783,E2 -31317.783} C_VEL
LIN {X 0,Y 54.484,Z 259.001,A -85,B 0,C 180,E1 -31318.661,E2 -31318.661} C_VEL
LIN {X 0,Y 46.025,Z 267.792,A -85,B 0,C 180,E1 -31319.998,E2 -31319.998} C_VEL
LIN {X 0,Y 38.666,Z 274.212,A -85,B 0,C 180,E1 -31321.29,E2 -31321.29} C_VEL
LIN {X 0,Y 28.232,Z 281.843,A -85,B 0,C 180,E1 -31325.233,E2 -31325.233} C_VEL
LIN {X 0,Y 18.035,Z 287.938,A -85,B 0,C 180,E1 -31333,E2 -31333} C_VEL
LIN {X 0,Y 8.921,Z 292.744,A -85,B 0,C 180,E1 -31357.993,E2 -31357.993} C_VEL
LIN {X 0,Y 6.366,Z 295.319,A -85,B 0,C 180,E1 -31409.977,E2 -31409.977} C_VEL
LIN {X 0,Y 9.117,Z 297.262,A -85,B 0,C 180,E1 -31460.408,E2 -31460.408} C_VEL
LIN {X 0,Y 21.447,Z 299.889,A -85,B 0,C 180,E1 -31489.409,E2 -31489.409} C_VEL
LIN {X 0,Y 28.268,Z 300.62,A -85,B 0,C 180,E1 -31493.924,E2 -31493.924} C_VEL
LIN {X 0,Y 28.143,Z 300.515,A -85,B 0,C 180,E1 -31497.203,E2 -31497.203} C_VEL
LIN {X 0,Y 21.092,Z 299.551,A -85,B 0,C 180,E1 -31501.814,E2 -31501.814} C_VEL
LIN {X 0,Y 14.285,Z 298.183,A -85,B 0,C 180,E1 -31510.324,E2 -31510.324} C_VEL
LIN {X 0,Y 6.294,Z 295.312,A -85,B 0,C 180,E1 -31556.092,E2 -31556.092} C_VEL
LIN {X 0,Y 10.413,Z 291.389,A -85,B 0,C 180,E1 -31632.467,E2 -31632.467} C_VEL
LIN {X 0,Y 20.006,Z 286.356,A -85,B 0,C 180,E1 -31651.443,E2 -31651.443} C_VEL
LIN {X 0,Y 30.221,Z 280.057,A -85,B 0,C 180,E1 -31658.483,E2 -31658.483} C_VEL
LIN {X 0,Y 40.588,Z 272.204,A -85,B 0,C 180,E1 -31662.254,E2 -31662.254} C_VEL
LIN {X 0,Y 47.302,Z 266.15,A -85,B 0,C 180,E1 -31663.834,E2 -31663.834} C_VEL
LIN {X 0,Y 50.618,Z 267.616,A -85,B 0,C 180,E1 -31664.478,E2 -31664.478} C_VEL
LIN {X 0,Y 50.618,Z 600,A -85,B 0,C 180,E1 -31664.478,E2 -31664.478} C_VEL
LIN {X 0,Y 50.618,Z 600,A -85,B 0,C 180,E1 -31664.478,E2 -31664.478}

QRS_NEXT_CUT()

QRS_NEXT()
QRS_HOME()

END
